// TwinCAT 3 PLC project Project_V25_Gr3
// ProgramVersion: 3.1.4026.13
// CompilerDefines: VISU_USEPROPERTYINFO
// libraries:
//   Tc2_Standard, * (Beckhoff Automation GmbH)
//   Tc2_System, * (Beckhoff Automation GmbH)
//   VisuDialogs, * (System)
// project tree:
//   / Engineer_HMI.TcVIS, GlobalTextList.TcGTLO, PlcTask.TcTTO, Visualization Manager.TcVMO (not stored)
//   Enums/ E_Status.TcDUT
//   Function Blocks/Currently not in use/ FB_EncoderScaling.TcPOU, FB_FeedForward.TcPOU (not stored), FB_Motion_Control.TcPOU, FB_SecondaryControlSinus.TcPOU, FB_SecondaryControlStartPos.TcPOU
//   Function Blocks/Deadband Comp/ FB_Deadband.TcPOU, FB_Deadband_Auto.TcPOU, FB_Deadband_Auto_sine.TcPOU
//   Function Blocks/Encoder_Payload/ FB_Encoder.TcPOU (not stored), FB_PayloadPosition.TcPOU
//   Function Blocks/FBs Auto Control/ FB_AutoSineMotion.TcPOU, FB_AutoStartPos.TcPOU, FB_Derivator.TcPOU, FB_SineActivation_SC.TcPOU
//   Function Blocks/FBs for Motion Control/Ekstra FBs/ FB_ControlReset_SC.TcPOU, FB_Feedforward_SC.TcPOU, FB_GainChooser.TcPOU (not stored), FB_Target_displacement.TcPOU
//   Function Blocks/FBs for Motion Control/ FB_Auto_Combination.TcPOU, FB_Auto_PC.TcPOU, FB_Auto_SC.TcPOU, FB_Enable_Motion.TcPOU, FB_EndStop.TcPOU, FB_Manual_PC.TcPOU, FB_Manual_SC.TcPOU, FB_MUX_selector.TcPOU, FB_Outputs.TcPOU
//   Function Blocks/ FB_Clock.TcPOU, FB_DisplacementControl.TcPOU, FB_DisplacementControl_SC.TcPOU, FB_DisplacementValveOutput.TcPOU, FB_Inputs.TcPOU, FB_Integrator.TcPOU, FB_Joystick.TcPOU, FB_StartPos.TcPOU, FB_StateMachine_Mode_Selection.TcPOU, FB_ValveOutput.TcPOU
//   Function Blocks/PIDgains/ FB_PIDgains.TcPOU
//   Function Blocks/Input_Scaling/ FB_JoystickInputScaling.TcPOU, FB_JoystickInputScaling_01.TcPOU (not stored), FB_PressureInputScaling.TcPOU (not stored), FB_Yoke_Input_Scaling.TcPOU (not stored)
//   Functions/ F_SineFunction_primary.TcPOU, F_SineFunction_secondary.TcPOU
//   GVLs/ G_IO.TcGVL, G_Motion_Control.TcGVL, G_Parameters.TcGVL, G_PID_Tuning.TcGVL, G_Sensors.TcGVL, G_Engineer_HMI.TcGVL
//   PIDs/ FB_PID_Controller.TcPOU, FB_PID_Controller_posref.TcPOU, FB_PID_controller_old.TcPOU, FB_PID_SC.TcPOU, FB_ResetIntegralController.TcPOU
//   POUs/ MAIN.TcPOU, P_MotionControl.TcPOU, P_Outputs.TcPOU
//   Structs/ ST_PressureInputScaling.TcDUT, ST_JoystickInputScaling.TcDUT, ST_Parameters.TcDUT, ST_ValveDeadBand.TcDUT, ST_ValveOutput.TcDUT, ST_YokeInputScaling.TcDUT
// real-time tasks:
//   TASK PlcTask: cycle T#10ms, priority 20, ADS port 350
// I/O:
//   DEVICE Device 1 (EtherCAT), AmsNetId 128.39.200.126.2.1
//     Term 1 (EK1200) [EK1200-5000 EtherCAT Power supply (2A E-Bus)]
//       Term 2 (EL1859) [EL1859 8Ch. Dig. Input 24V, 3ms, 8Ch. Dig. Output 24V, 0.5A]
//       Term 3 (EL3174) [EL3174 4Ch. Ana. Input +/-10V Diff., +/-20mA SingleEnded, 16 Bit]
//       Term 4 (EL4032) [EL4032 2Ch. Ana. Output +/-10V, 12bit]
//       Term 5 (EL3204) [EL3204 4Ch. Ana. Input PT100 (RTD)]
//       Term 6 (EK1110) [EK1110 EtherCAT extension]
//     Term 7 (EK1818) [EK1818 EtherCAT IO-Coupler  (1A E-Bus, 8 Ch. Dig. In, 3ms, 4 Ch. Dig. Out 24V, 0,5A)]
//       Term 8 (EL1008) [EL1008 8Ch. Dig. Input 24V, 3ms]
//       Term 9 (EL3174) [EL3174 4Ch. Ana. Input +/-10V Diff., +/-20mA SingleEnded, 16 Bit]
//       Term 10 (EL3068) [EL3068 8Ch. Ana. Input 0-10V]
//       Term 11 (EL4032) [EL4032 2Ch. Ana. Output +/-10V, 12bit]
//       Term 12 (EL4122) [EL4122 2Ch. Ana. Output  4-20mA, 16bit]
//       Term 14 (EL9011) [EL9011 End Terminal]
//     Box 13 (Fraba EtherCAT) [Absolute Rotary Encoder IXARC V01.05]
// variable links:
//   Project_V25_Gr3/Project_V25_Gr3 Instance <-> Device 1 (EtherCAT)/Box 13 (Fraba EtherCAT)
//     PlcTask Inputs/G_IO.nWinchEncoderValue <-> Encoder/Position Value
//   Project_V25_Gr3/Project_V25_Gr3 Instance <-> Device 1 (EtherCAT)/Term 7 (EK1818)
//     PlcTask Inputs/G_IO.bEmgOk <-> Channel 1/Input
//     PlcTask Outputs/G_IO.bEnablePCDV <-> Channel 10/Output
//     PlcTask Outputs/G_IO.bOpenBrakes <-> Channel 9/Output
//     PlcTask Outputs/G_IO.bWinchValveEnable <-> Channel 11/Output
//   Project_V25_Gr3/Project_V25_Gr3 Instance <-> Device 1 (EtherCAT)/Term 7 (EK1818)/Term 10 (EL3068)
//     PlcTask Inputs/G_IO.fJoyXraw <-> AI Standard Channel 6/Value
//     PlcTask Inputs/G_IO.fJoyYraw <-> AI Standard Channel 7/Value
//     PlcTask Inputs/G_IO.fJoyZraw <-> AI Standard Channel 8/Value
//     PlcTask Inputs/G_IO.fPressureReturn <-> AI Standard Channel 3/Value
//     PlcTask Inputs/G_IO.fPressureSupply <-> AI Standard Channel 2/Value
//     PlcTask Inputs/G_IO.fPressureWinchA <-> AI Standard Channel 1/Value
//     PlcTask Inputs/G_IO.fPressureWinchB <-> AI Standard Channel 4/Value
//   Project_V25_Gr3/Project_V25_Gr3 Instance <-> Device 1 (EtherCAT)/Term 7 (EK1818)/Term 11 (EL4032)
//     PlcTask Outputs/G_IO.fWinchPDCVOut <-> AO Outputs Channel 1/Analog output
//   Project_V25_Gr3/Project_V25_Gr3 Instance <-> Device 1 (EtherCAT)/Term 7 (EK1818)/Term 12 (EL4122)
//     PlcTask Outputs/G_IO.fWinchValveOut <-> Channel 1/Output
//   Project_V25_Gr3/Project_V25_Gr3 Instance <-> Device 1 (EtherCAT)/Term 7 (EK1818)/Term 8 (EL1008)
//     PlcTask Inputs/G_IO.bAutoSwitch <-> Channel 3/Input
//     PlcTask Inputs/G_IO.bDisplacementEnable <-> Channel 7/Input
//     PlcTask Inputs/G_IO.bManualSwitch <-> Channel 1/Input
//     PlcTask Inputs/G_IO.bOffSwitch <-> Channel 2/Input
//     PlcTask Inputs/G_IO.bStartButton <-> Channel 4/Input
//     PlcTask Inputs/G_IO.bStopButton <-> Channel 5/Input
//     PlcTask Inputs/G_IO.bWinchEnable <-> Channel 6/Input
//   Project_V25_Gr3/Project_V25_Gr3 Instance <-> Device 1 (EtherCAT)/Term 7 (EK1818)/Term 9 (EL3174)
//     PlcTask Inputs/G_IO.fPDCVMonitor <-> AI Standard Channel 1/Value
//     PlcTask Inputs/G_IO.fYoke <-> AI Standard Channel 4/Value
//     PlcTask Inputs/G_IO.nMoogMonitor <-> AI Standard Channel 2/Value

CONFIGURATION Project_V25_Gr3
    RESOURCE PLC ON TwinCAT3
        TASK PlcTask(INTERVAL := T#10ms, PRIORITY := 20);
        PROGRAM MAIN WITH PlcTask : MAIN;
    END_RESOURCE
END_CONFIGURATION

// ---- Enums/E_Status.TcDUT
{attribute 'qualified_only'}
{attribute 'strict'}
{attribute 'to_string'}
TYPE E_Status :
(
	Off,
	Fault,
	Ready,
	//Starting,
	Running,
	//Stopping,
	Checking
);
END_TYPE

// ---- Structs/ST_PressureInputScaling.TcDUT
TYPE ST_PressureInputScaling :
STRUCT
	fMaxInputValue 			: LREAL:= 32767.0;	// tunable max input value //   // denne verdien ble satt for å unngå å dele på 0, hvorfor må vi skrive det her men ikke i blueprint prosjekt
	fMinInputValue			: LREAL;	// tunable min input value  
	fMaxOutputValue  		: LREAL;	// max sensor output value
	fMinOutputValue  		: LREAL;	// min sensor output value	
END_STRUCT
END_TYPE

// ---- Structs/ST_JoystickInputScaling.TcDUT
TYPE ST_JoystickInputScaling :
STRUCT
	fMaxInputValue			: LREAL;	// tunable max input value
	fMinInputValue 			: LREAL;	// tunable min input value
	fNeutralInputValue  	: LREAL;	// tunable neutral input value
	fNeutralDeadband		: LREAL;	// tunable dead_band value
	fMaxOutputValue  		: LREAL;	// normalized max output value
	fMinOutputValue  		: LREAL;	// normalized min output value
	fNeutralOutputValue  	: LREAL;	// normalized neutral output value
END_STRUCT
END_TYPE

// ---- Structs/ST_Parameters.TcDUT
 TYPE ST_Parameters : // Blir gjort globale i GVL
STRUCT
	fCyclicTime 					: LREAL := 0.01; // [s]
	fMaxWinchVelocityLimit 			: LREAL := 0.25; // [m/s] Blueprint: 0.025
	fMaxWinchVelocityLimit_SC		: LREAL := 0.25;
	bWinchDeadBandCompOn 			: BOOL := FALSE;
	bDisplacementDeadBandCompOn 	: BOOL := FALSE;
	stWinchValveDeadBand 			: ST_ValveDeadBand := (fPosMax := 32767.0, fPosMin := 16383.0, fNegMin := 16383.0, fNegMax := 0.0);
	stDisplacementValveDeadBand 	: ST_ValveDeadBand := (fPosMax := 10000.0, fPosMin := 450.0, fNegMin := 450.0, fNegMax := 10000.0);
	stPressureSensorScaling400bar 	: ST_PressureInputScaling := (fMaxInputValue := 32767.0, fMinInputValue := 0.0, fMaxOutputValue := 400.0, fMinOutputValue := 0.0);
	stPressureSensorScaling40bar 	: ST_PressureInputScaling := (fMaxInputValue := 32767.0, fMinInputValue := 0.0, fMaxOutputValue := 40.0, fMinOutputValue := 0.0);
	stJoystickInputScalingX 		: ST_JoystickInputScaling := (fMaxInputValue := 14790.0, fMinInputValue := 1797.0, fNeutralInputValue := 8400, fNeutralDeadband := 50.0, fMaxOutputValue := 1.0, fMinOutputValue := 0.0, fNeutralOutputValue := 0.5);
	stJoystickInputScalingY 		: ST_JoystickInputScaling := (fMaxInputValue := 14770.0, fMinInputValue := 1829.0, fNeutralInputValue := 8340, fNeutralDeadband := 50.0, fMaxOutputValue := 1.0, fMinOutputValue := -1.0, fNeutralOutputValue := 0.0);
	stJoystickInputScalingZ 		: ST_JoystickInputScaling := (fMaxInputValue := 14830.0, fMinInputValue := 1804.0, fNeutralInputValue := 8380, fNeutralDeadband := 50.0, fMaxOutputValue := 1.0, fMinOutputValue := -1.0, fNeutralOutputValue := 0.0);
	fWinchEncoderOffset 			: LREAL := 12814.994735637447; // Encoder value at zero (Cylinder out / second layaer)
	stYokeInputScaling 				: ST_YokeInputScaling := (fMaxInputValue := 25000.0, fMinInputValue := 6150.0, fNeutralInputValue := 15470, fNeutralDeadband := 0.0, fMaxOutputValue := 1.0, fMinOutputValue := -1.0, fNeutralOutputValue := 0.0);
	fWinchDrumRadius 				: LREAL := 0.075;
	fWinchEndStopPos 				: LREAL := 3.0;
	fWinchEndStopPos_soft			: LREAL := 2.55;
	fWinchEndStopNeg 				: LREAL := 0.05;
	fWinchEndStopNeg_soft			: LREAL := 0.25;
	fPayloadMass 					: LREAL := 78.0;
	
	
END_STRUCT
END_TYPE

// ---- Structs/ST_ValveDeadBand.TcDUT
TYPE ST_ValveDeadBand :
STRUCT
	fPosMax	: LREAL; // Positive min value [19660..29490]
	fPosMin	: LREAL; // Positive max value [19660..29490]
	fNegMin : LREAL; // Negative max value [9830..19660]
	fNegMax	: LREAL; // Negative min value [9830..19660]
END_STRUCT
END_TYPE

// ---- Structs/ST_ValveOutput.TcDUT
TYPE ST_ValveOutput :
STRUCT
	bEnable					AT %Q* : BOOL := 0;
	nValveOutput 			AT %Q* : INT := 19660;
END_STRUCT
END_TYPE

// ---- Structs/ST_YokeInputScaling.TcDUT
TYPE ST_YokeInputScaling :
STRUCT
	fMaxInputValue			: LREAL;	// tunable max input value
	fMinInputValue 			: LREAL;	// tunable min input value
	fNeutralInputValue  	: LREAL;	// tunable neutral input value
	fNeutralDeadband		: LREAL;	// tunable dead_band value
	fMaxOutputValue  		: LREAL;	// normalized max output value
	fMinOutputValue  		: LREAL;	// normalized min output value
	fNeutralOutputValue  	: LREAL;	// normalized neutral output value
END_STRUCT
END_TYPE

// ---- GVLs/G_IO.TcGVL
{attribute 'qualified_only'}
VAR_GLOBAL
	// Digitale inputs
	bEmgOk 			     AT %I* : BOOL; 
	bStartButton 	     AT %I* : BOOL;
	bStopButton 	     AT %I* : BOOL; 
	bOffSwitch		     AT %I* : BOOL;  
	bManualSwitch	     AT %I* : BOOL; 
	bAutoSwitch		 	 AT %I* : BOOL; 
	bWinchEnable 		 AT %I* : BOOL; 
	bDisplacementEnable  AT %I* : BOOL;
	
	// Analoge Intputs
	fJoyXraw 			 AT %I* : INT; 
	fJoyYraw			 AT %I* : INT; 
	fJoyZraw 			 AT %I* : INT; 
	fPDCVMonitor		 AT %I* : INT; 
	nMoogMonitor		 AT %I* : INT; 
	fYoke				 AT %I* : INT; 
	fPressureWinchA 	 AT %I* : INT; 
	fPressureWinchB 	 AT %I* : INT; 
	fPressureSupply 	 AT %I* : INT; 
	fPressureReturn 	 AT %I* : INT; 
	nWinchEncoderValue	 AT %I* : UDINT; 
	
	// Digitale Outputs
	bOpenBrakes 		 AT %Q* : BOOL; 
	bEnablePCDV 		 AT %Q* : BOOL; 
	bWinchValveEnable 	 AT %Q* : BOOL; 
	
	// Analoge Outputs
	fWinchPDCVOut 		 AT %Q* : INT := 10000; 
	fWinchValveOut 		 AT %Q* : INT := 16383; 
	
	// New Test
	bTestNew AT %I* : BOOL;
	nTestNew AT %I* : INT;
	OutTestNew AT %Q* : BOOL;
	
END_VAR

// ---- GVLs/G_Motion_Control.TcGVL
{attribute 'qualified_only'}
VAR_GLOBAL
	//////////Primary Control/////////
//AutoStartPos
fWinchValveNormalizedInput 					: LREAL;	
bOpenBreak									: BOOL;

//AutoSineMotion
fWinchValveNormalizedInput_sine 			: LREAL;
fSineReferenceSignal						: LREAL;

// Position Errors
fPosition_error_SineMotion 					: LREAL; 
fPosition_error_StartPos					: LREAL;

//Displacement Sine
fDisplacementControlSignal_sine				: LREAL;

//Manual joystick posref
fWinchPosRefManual							: LREAL; //to make it a global variable for plotting 
fWinchValveInput_joystick_posref			: LREAL;



//////// Secondary control////////
fWinchPosRefManual_secondary				: LREAL;
fSCVInput_joystick_posref_secondary			: LREAL;

//Auto Sine Motion SC
fSineRefSignal_SC							: LREAL;
fVelRef_Sine_SC								: LREAL;

//Outer and inner loop sequence SC
fOutPutSignal_OL							: LREAL; //Skrive manual bak disse og oppdatere OPC UA
fDeadbandComp_out							: LREAL;

//Ikke lagt til i OPC UA
fOutPutSignal_OL_Auto						: LREAL;
fDeadbandComp_out_Auto						: LREAL;

//Ikke i bruk
fPosition_error_StartDisplacement 			: LREAL; 
fDisplacementControlSignal_Secondary		: LREAL;
bOpenBreak_Secondary						: BOOL;
END_VAR

// ---- GVLs/G_Parameters.TcGVL
{attribute 'qualified_only'}
VAR_GLOBAL
stParam		:	ST_Parameters;
END_VAR

// ---- GVLs/G_PID_Tuning.TcGVL
{attribute 'qualified_only'}
VAR_GLOBAL
	/////////Primary control/////////
	
	//MOOG valve
	fProportinalGain_output_MOOG 		: LREAL;
	fIntegralGain_output_MOOG			: LREAL;
	fDerivateGain_output_MOOG 			: LREAL;
	PID_output_MOOG						: LREAL;
	
	//Manual Control joystick pos ref
	fProportinalGain_output_joypos 		: LREAL;
	fIntegralGain_output_joypos			: LREAL;
	fDerivateGain_output_joypos 		: LREAL;
	ferror_joypos 						: LREAL;
	
	/////////Secondary control//////
	
	//Displacement control
	fYoke_error 						: LREAL;
	fPout_IL					 		: LREAL;
	fIout_IL					 		: LREAL;
	fDout_IL					 		: LREAL;
	PID_output_IL						: LREAL;
	Int_error_threshold					: LREAL := 0.0001;
	
	//Manual Control joystick posref secondary
	fPout_OL							: LREAL;
	fIout_OL							: LREAL;
	fDout_OL							: LREAL;
	fPout_OL_Auto							: LREAL;
	fIout_OL_Auto							: LREAL;
	fDout_OL_Auto							: LREAL;
	fPout_OL_Auto_sine							: LREAL;
	fIout_OL_Auto_sine							: LREAL;
	fDout_OL_Auto_sine							: LREAL;
	
	ferror_OL							: LREAL; //Skrive manual bak denne
	ferror_OL_Auto_startpos				: LREAL;
	ferror_OL_Auto_sine					: LREAL;
	
	
	////Combination////
	fPout_OL_combi							: LREAL;
	fIout_OL_combi							: LREAL;
	fDout_OL_combi							: LREAL;
	ferror_OL_combi							: LREAL;
	
END_VAR

// ---- GVLs/G_Sensors.TcGVL
{attribute 'qualified_only'}
VAR_GLOBAL
	fJoystickNormalizedY 					: LREAL; 
	fJoystickNormalizedX 					: LREAL; 
	fJoystickNormalizedZ 					: LREAL; 
	fYokeNormalizedFeedback 				: LREAL; 
	fPressureWinchA 	 					: LREAL; 
	fPressureWinchB 	 					: LREAL; 
	fPressureSupply 	 					: LREAL; 
	fPressureReturn 	 					: LREAL; 
	fWinchEncoderPosition 					: LREAL;
	fWinchEncoderPositionNormalized 		: LREAL;
	fPayLoadPosition 						: LREAL;
	fDeltaPMotor 							: LREAL;
	
	//Egentlig en Output/ NEIUNEI
	fWinchValveOutNormalized				: LREAL;
END_VAR

// ---- GVLs/G_Engineer_HMI.TcGVL
{attribute 'qualified_only'}
VAR_GLOBAL
	
//////////PID GAINS//////////

////Primary Control//////
// PID Manual control joystick pos ref Primary
	
	bPID_enable_JoyPosref_PC		: BOOL := TRUE;
	bPgain_enable_joy_posref		: BOOL := TRUE;
	bIgain_enable_joy_posref		: BOOL;
	bPgain_joy_posref_write			: BOOL;
	bIgain_joy_posref_write			: BOOL;
	bDgain_joy_posref_write			: BOOL;
	
	fPGain_JoyPosref_PC 			: LREAL;
	fIGain_JoyPosref_PC				: LREAL;
	fDGain_JoyPosref_PC				: LREAL;

// PID MOOG Valve (Auto PC)
	fPgain_MOOG						: LREAL;
	bPenable_MOOG					: BOOL := TRUE; //Ønsker P ledd på fra start
	bPgain_MOOG_write				: BOOL;
	
	fIgain_MOOG 					: LREAL; 
	bIenable_MOOG 					: BOOL;
	bIgain_MOOG_write				: BOOL; 

////// Secondary Control ////////

// PID Outer loop 
bPID_enable_OL					: BOOL := TRUE;

fPGain_OL_Pos					: LREAL;
fPGain_OL_Neg					: LREAL;
bPenable_OL						: BOOL := TRUE;
bPGain_OL_write_pos				: BOOL;
bPGain_OL_write_neg				: BOOL;

fIGain_OL_Pos					: LREAL;
fIGain_OL_Neg					: LREAL;
bIenable_OL						: BOOL;
bIGain_OL_write_pos				: BOOL;
bIGain_OL_write_neg				: BOOL;

// PID Inner loop
bPID_enable_IL					: BOOL := TRUE;

fPGain_IL_Pos					: LREAL;
fPGain_IL_Neg					: LREAL;
bPenable_IL						: BOOL := TRUE;
bPGain_IL_write_pos				: BOOL;
bPGain_IL_write_neg				: BOOL;

fIGain_IL_Pos					: LREAL;
fIGain_IL_Neg					: LREAL;
bIenable_IL						: BOOL;
bIGain_IL_write_pos				: BOOL;
bIGain_IL_write_neg				: BOOL;

fDGain_IL_Pos					: LREAL;
fDGain_IL_Neg					: LREAL;
bDenable_IL						: BOOL;
bDGain_IL_write_pos					: BOOL;
bDGain_IL_write_neg					: BOOL;



////////// PID GAINS End ///////////////////


	//Control chooser
	bPrimary_Control				: BOOL;	
	bPrimary_Control_active			: BOOL := FALSE;
	bSecondary_Control				: BOOL;
	bSecondary_Control_active		: BOOL := FALSE;

	//Endstop
	bEndStopUpActive 				: BOOL;
	bEndStopDownActive 				: BOOL;
	bEndStopOverride 				: BOOL; 
	
	/////Primary Control//////
	bManualControl_enable			: BOOL;
	
	
	
	// Auto Start Pos
	bAutoStartPosEnable				: BOOL;
	fAutoStartPos_target			: LREAL := 1.4;
	
	// Auto Sine Motion
	bAutoSineMotionEnable			 : BOOL; 
	
	// Displacement Sine Wave control: 
	bSineDisplacement				 : BOOL; 
	
	//Sine wave parameters
	fAmp 							: LREAL := 0.2;
	fFreq 							: LREAL := 0.1;
	fSinemidpoint					: LREAL := 1.4;
	ft_ENV							: LREAL := 10.0;
	
	
	
	
///// Primary Control End///////	
	
	
////// Secondary Control///////
	
//Displacementcontrol 
	bDisplacement_target_active		: BOOL;
	fDisplacement_target			: LREAL := 1.0;
	bJoystick_slider_active			: BOOL;
	bSecondaryStartPosEnable 		: BOOL;
	fSecondaryStartPos_target		: LREAL := 1.4;
	bSecondarySineMotionEnable		: BOOL;


	
	//Integral reset (antiwindup)
	fMaxerror_dis					: LREAL;
	
	
//PID Gains for Manual control joystick posref
	
	bManual_Secondary_joyposref_enable	: BOOL := TRUE;
	
// Deadband compensation (gjort om til var persistants som ligger i FB_PIDgains)
fUpperdeadband						: LREAL;
fNeutraldeadband					: LREAL;
fLowerdeadband						: LREAL;
bUpperWrite							: BOOL;
bNeutralWrite						: BOOL;
bLowerWrite							: BOOL;
	
////////Primary and Secondary combination//////
bCombinationActive					: BOOL;
bAutoSineCombi						: BOOL;

	
//StepInput displacement ikke lagt inn etter å ha ryddet, kan legges inn i 
//Manual SC om det trengs (la tidligere i P_outputs
bStepInput								: BOOL;
bStartStepInput							: BOOL;
fStepInput								: LREAL;
fDuration								: LREAL;

	
END_VAR

// ---- POUs/MAIN.TcPOU
PROGRAM MAIN
VAR
	bFunction_Blocks_enable				: BOOL := TRUE;
	fb_StateMachine_Mode_Selection	 	: FB_StateMachine_Mode_Selection;
	fb_Joystick_input_Scaling			: FB_JoystickInputScaling;
	fb_Joystick							: FB_Joystick;
	fb_ValveOutput						: FB_ValveOutput;
	fb_Encoder							: FB_Encoder; 
	fb_PressureInputScaling 			: FB_PressureInputScaling;
	fb_PayloadPosition					: FB_PayloadPosition;
	fb_Inputs							: FB_Inputs;
	eStatus								: E_Status;
	
	fbPIDgains							: FB_PIDgains;
END_VAR

P_MotionControl();

IF bFunction_Blocks_enable THEN
	fb_StateMachine_Mode_Selection();
	fb_Joystick_input_Scaling();
	fb_Joystick();
	fb_ValveOutput();
	fb_Encoder();
	fb_PressureInputScaling();
	fb_PayloadPosition();
	fb_Inputs();
	
	fbPIDgains();
END_IF

//Update eStatus
fb_StateMachine_Mode_Selection(
	eStatus => eStatus
	);
//	eStatus := E_Status.Running;
	
	

////////Select Primary eller Secondary control//////////////
IF G_Engineer_HMI.bPrimary_Control THEN
	G_Engineer_HMI.bPrimary_Control_active := TRUE;
	G_Engineer_HMI.bSecondary_Control_active := FALSE;
ELSIF G_Engineer_HMI.bSecondary_Control THEN
	G_Engineer_HMI.bPrimary_Control_active := FALSE;
	G_Engineer_HMI.bSecondary_Control_active := TRUE;
END_IF

END_PROGRAM

// ---- Function Blocks/FB_StateMachine_Mode_Selection.TcPOU
FUNCTION_BLOCK FB_StateMachine_Mode_Selection
VAR_INPUT
END_VAR
VAR_OUTPUT
eStatus : E_Status := E_Status.Checking; //Er dette til for å definere utgangen, kunne vi brukt structen (Enumen) direkte i koden?
END_VAR
VAR
	
	bStatusOk : BOOL; // Control variable 
	bFault : BOOL := FALSE;
	//bRunning : BOOL := TRUE; ikke nødvendig
END_VAR

	// State Machine for mode selection - Off, Fault, Ready, Running and Checking 
	
	// Variable bStatusOk, used troughout the function: 
IF G_IO.bEmgOk AND NOT(G_IO.bStopButton) AND NOT(G_IO.bOffSwitch) AND NOT(bFault) THEN 
	bStatusOk := TRUE;
ELSE 
	bStatusOk := FALSE;
END_IF

CASE eStatus OF
	E_Status.Checking: // Checking state (initially here)
	  IF bFault THEN
         eStatus := E_Status.Fault; 
	  END_IF
	  
	  IF bStatusOk THEN 
		  eStatus := E_Status.Ready;
	  END_IF
	  
	  IF NOT bStatusOk THEN
		 eStatus := E_Status.Off;
	  END_IF
	  
	 E_Status.Off:
	   IF bStatusOk THEN
			eStatus := E_Status.Checking;
	END_IF
		
	IF bFault THEN
			eStatus := E_Status.Fault;
	END_IF
		
	  E_Status.Fault:
		  IF NOT bFault THEN
			  eStatus := E_Status.Checking;
		  END_IF
		  
	E_Status.Ready:
	  IF G_IO.bStartButton AND bStatusOk THEN 
		  eStatus := E_Status.Running;
	  END_IF
	  
	  IF NOT(bStatusOk) OR bFault THEN
		  eStatus := E_Status.Checking;
	  END_IF
	  
	E_Status.Running: 
	
	 IF NOT(bStatusOk) OR bFault THEN 
		 eStatus := E_Status.Checking;
	 END_IF
	 
	 ELSE 
		 eStatus := E_Status.Checking;
  END_CASE

END_FUNCTION_BLOCK

// ---- Function Blocks/Input_Scaling/FB_JoystickInputScaling.TcPOU
FUNCTION_BLOCK FB_JoystickInputScaling
VAR_INPUT
	bEnable 				: BOOL;
	nRawInput 				: INT;
	stJoystickInputScaling  : ST_JoystickInputScaling;
END_VAR
VAR_OUTPUT
	fNormalizedOutput 		: LREAL;
END_VAR
VAR
	fRawInput 				: LREAL;
	fTempInput 				: LREAL;
	fTempOutput 			: LREAL;
END_VAR

fRawInput := INT_TO_LREAL(nRawInput);

fTempInput := fRawInput - stJoystickInputScaling.fNeutralInputValue;

IF fTempInput > stJoystickInputScaling.fNeutralDeadband THEN
	fTempOutput := fTempInput/(stJoystickInputScaling.fMaxInputValue - stJoystickInputScaling.fNeutralInputValue);
ELSIF fTempInput < -stJoystickInputScaling.fNeutralDeadband THEN	
	fTempOutput := fTempInput/(stJoystickInputScaling.fNeutralInputValue - stJoystickInputScaling.fMinInputValue);
ELSE
	fTempOutput := 0.0;
END_IF

IF NOT(bEnable) THEN
	fNormalizedOutput := 0.0;
ELSE
	fNormalizedOutput := LIMIT(stJoystickInputScaling.fMinOutputValue, fTempOutput, stJoystickInputScaling.fMaxOutputValue);
END_IF

END_FUNCTION_BLOCK

// ---- Function Blocks/FB_Joystick.TcPOU
FUNCTION_BLOCK FB_Joystick
VAR_INPUT
	bEnable 			: BOOL;
	fNormalizedInput 	: LREAL;
	stParam 			: ST_Parameters;
END_VAR
VAR_OUTPUT
	fOuput : LREAL;
END_VAR
VAR
END_VAR

IF bEnable THEN
	
	fOuput := fNormalizedInput*G_Parameters.stParam.fMaxWinchVelocityLimit_SC;
ELSE
	fOuput := 0.0;
END_IF

END_FUNCTION_BLOCK

// ---- Function Blocks/FB_ValveOutput.TcPOU
FUNCTION_BLOCK FB_ValveOutput
VAR_INPUT
	bEnable : BOOL; 
	bDeadBandCompOn : BOOL;
	stValveDeadBand : ST_ValveDeadBand; 
	fNormalizedInput : LREAL; 
END_VAR
VAR_OUTPUT
	bEnableValveOutput : BOOL; 
	nOutput : INT; 
END_VAR
VAR
	nOffset 	: INT := 16383; // KVIFOR
	nMaxValue	: INT := 20000;
	nMinValue 	: INT :=  12766;
	nTempOutput : INT := 16383;
END_VAR

//To måter er satt opp, kan endres i Engineer_HMI. En er satte parametere, den andre er parametere fra struct
IF bDeadBandCompOn THEN
	IF fNormalizedInput > 0.0 THEN
		nTempOutput := LREAL_TO_INT(ABS(fNormalizedInput*(stValveDeadBand.fPosMax - stValveDeadBand.fPosMin) + stValveDeadBand.fPosMin));
	ELSIF fNormalizedInput < 0.0 THEN 
		nTempOutput := LREAL_TO_INT(ABS(fNormalizedInput*(stValveDeadBand.fNegMax - stValveDeadBand.fNegMin) - stValveDeadBand.fNegMin));	
	ELSE 
		nTempOutput := nOffset;	//Offset ses som 0 (nøytral), fordi signalet går fra 0 til 32767.												
	END_IF

ELSE 
	IF fNormalizedInput > 0.0  THEN
		//Gjør om inputen mellom 0 og 1 til en output mellom 16383 (nøytral) og 32767(max)
		nTempOutput := LREAL_TO_INT(ABS(fNormalizedInput*(32767.0 - 16383.0) + 16383.0)); //ABS må til fordi output er en positiv verdi mellom 0 og 32767
	ELSIF fNormalizedInput < 0.0  THEN
		//Gjør om inputen mellom 0 og -1 til en output mellom 0 (min) og 16383 (nøytral)
		nTempOutput := LREAL_TO_INT(ABS(fNormalizedInput*(0 - 16383.0) - 16383.0));
	ELSE
		nTempOutput := nOffset; //Her settes også verdien til nøytral om det ikke er noen input
	END_IF	
	
END_IF

//Om den er enabled blir verdien sendt ut
IF bEnable THEN
	
	nOutput := LIMIT(nMinValue, nTempOutput, nMaxValue);
	bEnableValveOutput := TRUE;
//Eller så sender den ut nøytral verdi
ELSE 
	nOutput := nOffset;
	bEnableValveOutput := FALSE;
END_IF

END_FUNCTION_BLOCK

// ---- Function Blocks/Encoder_Payload/FB_PayloadPosition.TcPOU
FUNCTION_BLOCK FB_PayloadPosition
VAR_INPUT
END_VAR
VAR_OUTPUT
END_VAR
VAR
END_VAR

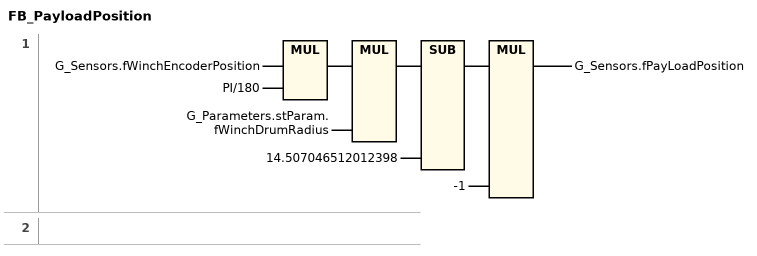
// NETWORK 1
G_Sensors.fPayLoadPosition := ((G_Sensors.fWinchEncoderPosition * (PI/180)) * G_Parameters.stParam.fWinchDrumRadius - 14.507046512012398) * -1;

// NETWORK 2

END_FUNCTION_BLOCK

// ---- Function Blocks/FB_Inputs.TcPOU
FUNCTION_BLOCK FB_Inputs 
VAR_INPUT
	fbJoystickWinch : FB_JoystickInputScaling; 
	fbJoystickRot : FB_JoystickInputScaling; 
	fbYokeInputScaling : FB_Yoke_Input_Scaling;
	fbWinchPosition : FB_Encoder;
	fbPressureSupply : FB_PressureInputScaling; 
	fbPressureReturn : FB_PressureInputScaling;
	fbPressureWinch_A_Input : FB_PressureInputScaling;
	fbPressureWInch_B_Input : FB_PressureInputScaling; 
END_VAR
VAR_OUTPUT
END_VAR
VAR
END_VAR

fbJoystickWinch(
	bEnable := G_IO.bAutoSwitch OR G_IO.bManualSwitch,
	nRawInput := G_IO.fJoyYraw, 
	stJoystickInputScaling := G_Parameters.stParam.stJoystickInputScalingY, 
	fNormalizedOutput => G_Sensors.fJoystickNormalizedY
);

fbJoystickRot(
	bEnable := G_IO.bManualSwitch, 
	nRawInput := G_IO.fJoyZraw,
	stJoystickInputScaling := G_Parameters.stParam.stJoystickInputScalingZ,
    fNormalizedOutput => G_Sensors.fJoystickNormalizedZ
);

fbYokeInputScaling(
	bEnable := TRUE, //Vil lese Yokeverdi hele tiden så den settes til TRUE (var G_IO.bManualSwitch før)
	nRawInput := G_IO.fYoke, 
	stYokeInputScaling := G_Parameters.stParam.stYokeInputScaling,
	fNormalizedOutput => G_Sensors.fYokeNormalizedFeedback
);

fbWinchPosition(
nRawInput := G_IO.nWinchEncoderValue,
fEncoderOffset := G_Parameters.stParam.fWinchEncoderOffset,
fPosition => G_Sensors.fWinchEncoderPosition
);

fbPressureSupply(
	nRawInput := G_IO.fPressureSupply,
	stPressureInputScaling := G_Parameters.stParam.stPressureSensorScaling400bar,
	fOutput => G_Sensors.fPressureSupply
);

fbPressureReturn(
	nRawInput := G_IO.fPressureReturn,
	stPressureInputScaling := G_Parameters.stParam.stPressureSensorScaling40bar,
	fOutput => G_Sensors.fPressureReturn
	);
	
fbPressureWinch_A_Input(
	nRawInput := G_IO.fPressureWinchA, 
	stPressureInputScaling := G_Parameters.stParam.stPressureSensorScaling400bar, 
	fOutput => G_Sensors.fPressureWinchA
	);
	
fbPressureWinch_B_Input(
nRawInput := G_IO.fPressureWinchB,
stPressureInputScaling := G_Parameters.stParam.stPressureSensorScaling400bar, 
fOutput => G_Sensors.fPressureWinchB
);

// Trykkfall over motor: 

G_Sensors.fDeltaPMotor := (G_Sensors.fPressureWinchA - G_Sensors.fPressureWinchB);

END_FUNCTION_BLOCK

// ---- Function Blocks/PIDgains/FB_PIDgains.TcPOU
FUNCTION_BLOCK FB_PIDgains
VAR_INPUT
END_VAR
VAR_OUTPUT
END_VAR

VAR PERSISTENT
	
	/////Primary Control/////
	
	//Joystick Posref
	fPGain_JoyPosref_PC 				: LREAL;
	fIGain_JoyPosref_PC					: LREAL;
	fDGain_JoyPosref_PC					: LREAL;
	
	
	//Auto PC
	fPGain_MOOG							: LREAL;
	fIGain_MOOG							: LREAL;
	
	/////Secondary Control////
	
	//Outer loop
	fPGain_OL_Pos					: LREAL;
	fIGain_OL_Pos					: LREAL;
	fPGain_OL_Neg					: LREAL;
	fIGain_OL_Neg					: LREAL;
	
	//Inner loop
	fPGain_IL_Pos					: LREAL;
	fIGain_IL_Pos					: LREAL;
	fPGain_IL_Neg					: LREAL;
	fIGain_IL_Neg					: LREAL;
	fDGain_IL_Pos					: LREAL;
	fDGain_IL_Neg					: LREAL;
	
	/////Deadband Compensation/////
	fUpper							: LREAL;
	fNeutral						: LREAL;
	fLower							: LREAL;
	
END_VAR

VAR
END_VAR

	
	/////Primary Control/////
	
	//Joystick Posref
IF NOT(G_Engineer_HMI.bPgain_joy_posref_write) THEN
	G_Engineer_HMI.fPGain_JoyPosref_PC := fPGain_JoyPosref_PC; //Update to the persistent variable
ELSE
	fPGain_JoyPosref_PC := G_Engineer_HMI.fPGain_JoyPosref_PC; //Connect the gain to the global HMI
END_IF
	
	
IF NOT(G_Engineer_HMI.bIgain_joy_posref_write) THEN
	G_Engineer_HMI.fIGain_JoyPosref_PC := fIGain_JoyPosref_PC; //Update to the persistent variable
ELSE
	fIGain_JoyPosref_PC := G_Engineer_HMI.fIGain_JoyPosref_PC; //Connect the gain to the global HMI
END_IF
	
	
IF NOT(G_Engineer_HMI.bDgain_joy_posref_write) THEN
	G_Engineer_HMI.fDGain_JoyPosref_PC := fDGain_JoyPosref_PC; //Update to the persistent variable
ELSE
	fDGain_JoyPosref_PC := G_Engineer_HMI.fDGain_JoyPosref_PC; //Connect the gain to the global HMI
END_IF
	
	//Auto PC
IF NOT(G_Engineer_HMI.bPgain_MOOG_write) THEN
	G_Engineer_HMI.fPgain_MOOG := fPGain_MOOG; 
ELSE
	fPGain_MOOG := G_Engineer_HMI.fPgain_MOOG;
END_IF


IF NOT(G_Engineer_HMI.bIgain_MOOG_write) THEN
	G_Engineer_HMI.fIgain_MOOG := fIGain_MOOG;
ELSE
	fIGain_MOOG := G_Engineer_HMI.fIgain_MOOG;
END_IF	


//////// Secondary Control /////////

//Outer loop
//Positive
IF NOT(G_Engineer_HMI.bPGain_OL_write_pos) THEN
	G_Engineer_HMI.fPGain_OL_Pos := fPGain_OL_Pos; 
ELSE
	fPGain_OL_Pos := G_Engineer_HMI.fPGain_OL_Pos;
END_IF


IF NOT(G_Engineer_HMI.bIGain_OL_write_pos) THEN
	G_Engineer_HMI.fIGain_OL_Pos := fIGain_OL_Pos;
ELSE
	fIGain_OL_Pos := G_Engineer_HMI.fIGain_OL_Pos;
END_IF	

//Negative
IF NOT(G_Engineer_HMI.bPGain_OL_write_neg) THEN
	G_Engineer_HMI.fPGain_OL_Neg := fPGain_OL_Neg; 
ELSE
	fPGain_OL_Neg := G_Engineer_HMI.fPGain_OL_Neg;
END_IF


IF NOT(G_Engineer_HMI.bIGain_OL_write_neg) THEN
	G_Engineer_HMI.fIGain_OL_Neg := fIGain_OL_Neg;
ELSE
	fIGain_OL_Neg := G_Engineer_HMI.fIGain_OL_Neg;
END_IF	


//Inner loop
//Positive
IF NOT(G_Engineer_HMI.bPGain_IL_write_pos) THEN
	G_Engineer_HMI.fPGain_IL_Pos := fPGain_IL_Pos; 
ELSE
	fPGain_IL_Pos := G_Engineer_HMI.fPGain_IL_Pos;
END_IF


IF NOT(G_Engineer_HMI.bIGain_IL_write_pos) THEN
	G_Engineer_HMI.fIGain_IL_Pos := fIGain_IL_Pos;
ELSE
	fIGain_IL_Pos := G_Engineer_HMI.fIGain_IL_Pos;
END_IF	

IF NOT(G_Engineer_HMI.bDGain_IL_write_pos) THEN
	G_Engineer_HMI.fDGain_IL_Pos := fDGain_IL_Pos;
ELSE
	fDGain_IL_Pos := G_Engineer_HMI.fDGain_IL_Pos;
END_IF	

//Negative
IF NOT(G_Engineer_HMI.bPGain_IL_write_neg) THEN
	G_Engineer_HMI.fPGain_IL_Neg := fPGain_IL_Neg; 
ELSE
	fPGain_IL_Neg := G_Engineer_HMI.fPGain_IL_Neg;
END_IF


IF NOT(G_Engineer_HMI.bIGain_IL_write_neg) THEN
	G_Engineer_HMI.fIGain_IL_Neg := fIGain_IL_Neg;
ELSE
	fIGain_IL_Neg := G_Engineer_HMI.fIGain_IL_Neg;
END_IF	

IF NOT(G_Engineer_HMI.bDGain_IL_write_neg) THEN
	G_Engineer_HMI.fDGain_IL_Neg := fDGain_IL_Neg;
ELSE
	fDGain_IL_Neg := G_Engineer_HMI.fDGain_IL_Neg;
END_IF	

/////////Deadband Compensation////////////
IF NOT(G_Engineer_HMI.bUpperWrite) THEN
	G_Engineer_HMI.fUpperdeadband := fUpper;
ELSE
	fUpper := G_Engineer_HMI.fUpperdeadband;
END_IF

IF NOT(G_Engineer_HMI.bNeutralWrite) THEN
	G_Engineer_HMI.fNeutraldeadband := fNeutral;
ELSE
	fNeutral := G_Engineer_HMI.fNeutraldeadband;
END_IF

IF NOT(G_Engineer_HMI.bLowerWrite) THEN
	G_Engineer_HMI.fLowerdeadband:= fLower;
ELSE
	fLower := G_Engineer_HMI.fLowerdeadband;
END_IF

END_FUNCTION_BLOCK

// ---- POUs/P_MotionControl.TcPOU
PROGRAM P_MotionControl
VAR
	

//////Dette brukes i det nye////////////

//Enable Motion
	bAutoEnable_PC 							: BOOL;
	bManualEnable_PC 						: BOOL; 
	bAutoEnable_SC 							: BOOL; 
	bManualEnable_SC					    : BOOL;
	bCombinationEnable						: BOOL;

/////////// Function blocks////////// 
	
	//Enable Motion
	fbEnableMotion							: FB_Enable_Motion;
	
	//Primary Control
	fbManual_PC								: FB_Manual_PC;
	fbAuto_PC								: FB_Auto_PC;
	
	//Secondary Control
	fbManual_SC								: FB_Manual_SC;
	fbAuto_SC								: FB_Auto_SC;

	//Combination
	fbCombination							: FB_Auto_Combination;

	//Endstop
	fbEndstop								: FB_EndStop;

	//MUX
	fbMUX_selector							: FB_MUX_selector;

/////OutPut Variables////
	fPCV_MPC							: LREAL;
	fSCV_MPC							: LREAL;
	
	fPCV_APC							: LREAL;
	fSCV_APC							: LREAL;
	
	fPCV_MSC							: LREAL;
	fSCV_MSC							: LREAL;
	
	fPCV_ASC							: LREAL;
	fSCV_ASC							: LREAL;
	
	fPCV_combi							: LREAL;
	fSCV_combi							: LREAL;
	
	//After MUX
	fPCV							: LREAL;
	fSCV							: LREAL;
	fPCV_norm_input					: LREAL;
	fSCV_norm_input					: LREAL;
	
	
//ValveOutputs
fbOutputs							: FB_Outputs;
fPCV_raw							: INT;
fSCV_raw							: INT;
	
END_VAR

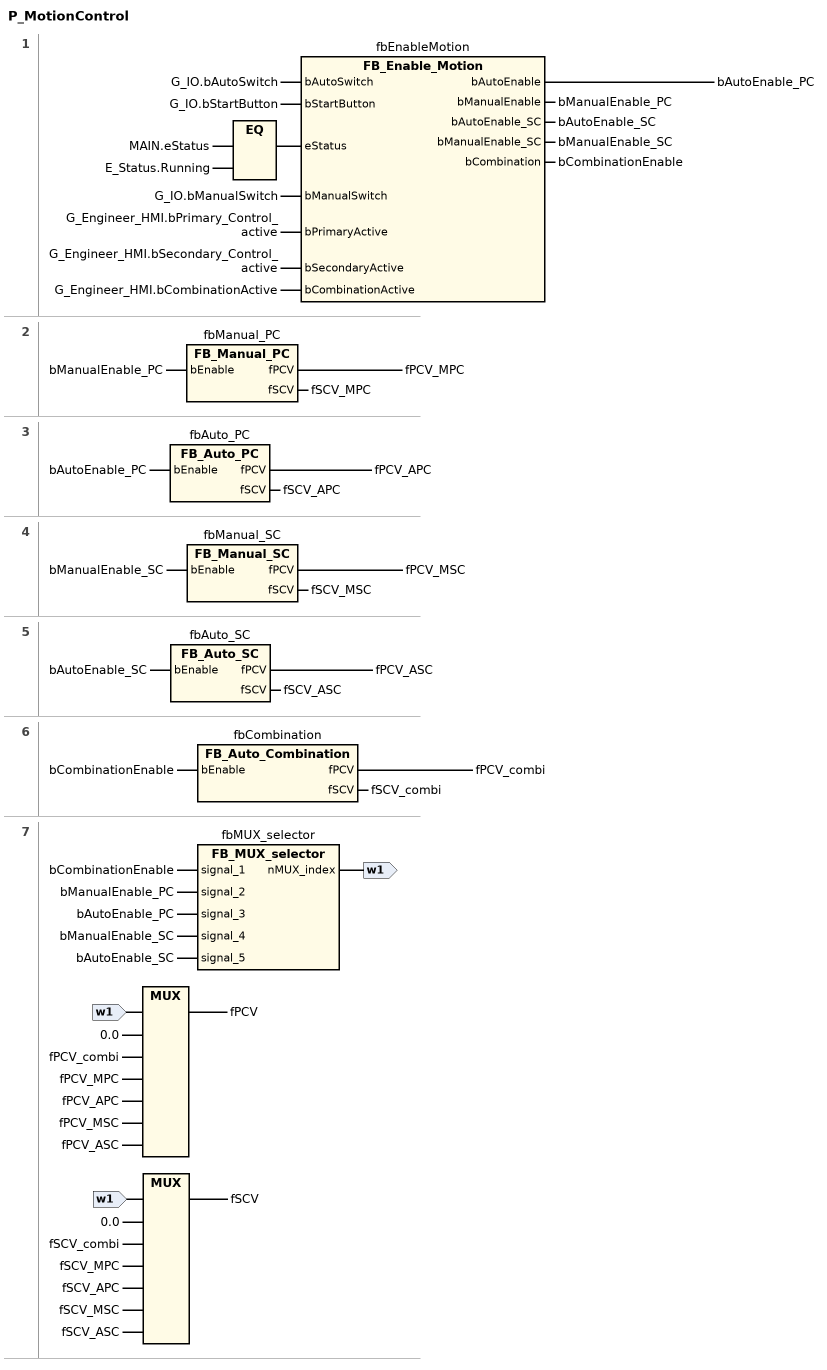
// NETWORK 1
fbEnableMotion(
    bAutoSwitch := G_IO.bAutoSwitch,
    bStartButton := G_IO.bStartButton,
    eStatus := MAIN.eStatus = E_Status.Running,
    bManualSwitch := G_IO.bManualSwitch,
    bPrimaryActive := G_Engineer_HMI.bPrimary_Control_active,
    bSecondaryActive := G_Engineer_HMI.bSecondary_Control_active,
    bCombinationActive := G_Engineer_HMI.bCombinationActive,
    bManualEnable => bManualEnable_PC,
    bAutoEnable_SC => bAutoEnable_SC,
    bManualEnable_SC => bManualEnable_SC,
    bCombination => bCombinationEnable); // FB_Enable_Motion
bAutoEnable_PC := fbEnableMotion.bAutoEnable;

// NETWORK 2
fbManual_PC(bEnable := bManualEnable_PC, fSCV => fSCV_MPC); // FB_Manual_PC
fPCV_MPC := fbManual_PC.fPCV;

// NETWORK 3
fbAuto_PC(bEnable := bAutoEnable_PC, fSCV => fSCV_APC); // FB_Auto_PC
fPCV_APC := fbAuto_PC.fPCV;

// NETWORK 4
fbManual_SC(bEnable := bManualEnable_SC, fSCV => fSCV_MSC); // FB_Manual_SC
fPCV_MSC := fbManual_SC.fPCV;

// NETWORK 5
fbAuto_SC(bEnable := bAutoEnable_SC, fSCV => fSCV_ASC); // FB_Auto_SC
fPCV_ASC := fbAuto_SC.fPCV;

// NETWORK 6
fbCombination(bEnable := bCombinationEnable, fSCV => fSCV_combi); // FB_Auto_Combination
fPCV_combi := fbCombination.fPCV;

// NETWORK 7
fbMUX_selector(
    signal_1 := bCombinationEnable,
    signal_2 := bManualEnable_PC,
    signal_3 := bAutoEnable_PC,
    signal_4 := bManualEnable_SC,
    signal_5 := bAutoEnable_SC); // FB_MUX_selector
fPCV := MUX(fbMUX_selector.nMUX_index, 0.0, fPCV_combi, fPCV_MPC, fPCV_APC, fPCV_MSC, fPCV_ASC);
fSCV := MUX(fbMUX_selector.nMUX_index, 0.0, fSCV_combi, fSCV_MPC, fSCV_APC, fSCV_MSC, fSCV_ASC);

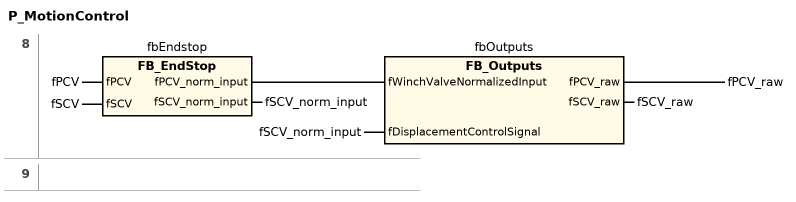
// NETWORK 8
fbEndstop(fPCV := fPCV, fSCV := fSCV, fSCV_norm_input => fSCV_norm_input); // FB_EndStop
fbOutputs(
    fWinchValveNormalizedInput := fbEndstop.fPCV_norm_input,
    fDisplacementControlSignal := fSCV_norm_input,
    fSCV_raw => fSCV_raw); // FB_Outputs
fPCV_raw := fbOutputs.fPCV_raw;

// NETWORK 9

END_PROGRAM

// ---- Function Blocks/FBs for Motion Control/FB_Enable_Motion.TcPOU
FUNCTION_BLOCK FB_Enable_Motion
VAR_INPUT
	bAutoSwitch								: BOOL;
	bStartButton							: BOOL;
	
	eStatus									: BOOL;
	
	bManualSwitch							: BOOL;
	
	bPrimaryActive							: BOOL;
	bSecondaryActive						: BOOL;
	bCombinationActive						: BOOL;
	
END_VAR
VAR_OUTPUT
	bAutoEnable 							: BOOL;
	bManualEnable 							: BOOL; 
	bAutoEnable_SC 							: BOOL; 
	bManualEnable_SC					    : BOOL;
	bCombination							: BOOL;
END_VAR
VAR
END_VAR

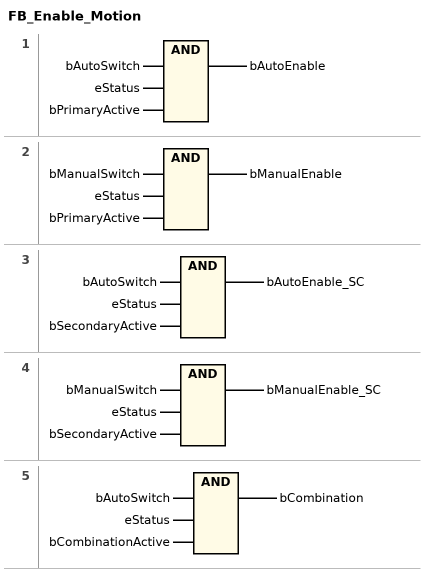
// NETWORK 1
bAutoEnable := bAutoSwitch AND eStatus AND bPrimaryActive;

// NETWORK 2
bManualEnable := bManualSwitch AND eStatus AND bPrimaryActive;

// NETWORK 3
bAutoEnable_SC := bAutoSwitch AND eStatus AND bSecondaryActive;

// NETWORK 4
bManualEnable_SC := bManualSwitch AND eStatus AND bSecondaryActive;

// NETWORK 5
bCombination := bAutoSwitch AND eStatus AND bCombinationActive;

END_FUNCTION_BLOCK

// ---- Function Blocks/FBs for Motion Control/FB_Manual_PC.TcPOU
FUNCTION_BLOCK FB_Manual_PC
VAR_INPUT
	bEnable					: BOOL;
END_VAR
VAR_OUTPUT
	fPCV					: LREAL;
	fSCV					: LREAL;
END_VAR
VAR
	//Function Blocks
	fbJoystick				: FB_Joystick;
	fbGetStartPos			: FB_StartPos;
	fbWinchVelIntegrator	: FB_Integrator;
	fbPID_Controller		: FB_PID_Controller;
	fbMUX_selector			: FB_MUX_selector;
	
	//Manual PosRef
	fWinchVelRefManual		: LREAL;
	fWInchVelRefAuto		: LREAL; //Brukes ikke
	fInitialWinchPos		: LREAL;
	
	//Valve signals
	fPCV_Manual			: LREAL;
	fPCV_PosRef			: LREAL;
	fPCV_Off			: LREAL;
	fSCV_On				: LREAL;
	fSCV_Off			: LREAL;
	
	
	//Notat på hva som skal til OPC UA
	//G_Motion_Control.fWinchPosRefManual
	


	END_VAR
VAR // added by the converter: edge detectors and wires of the graphical bodies
    _w1 : BOOL;
END_VAR

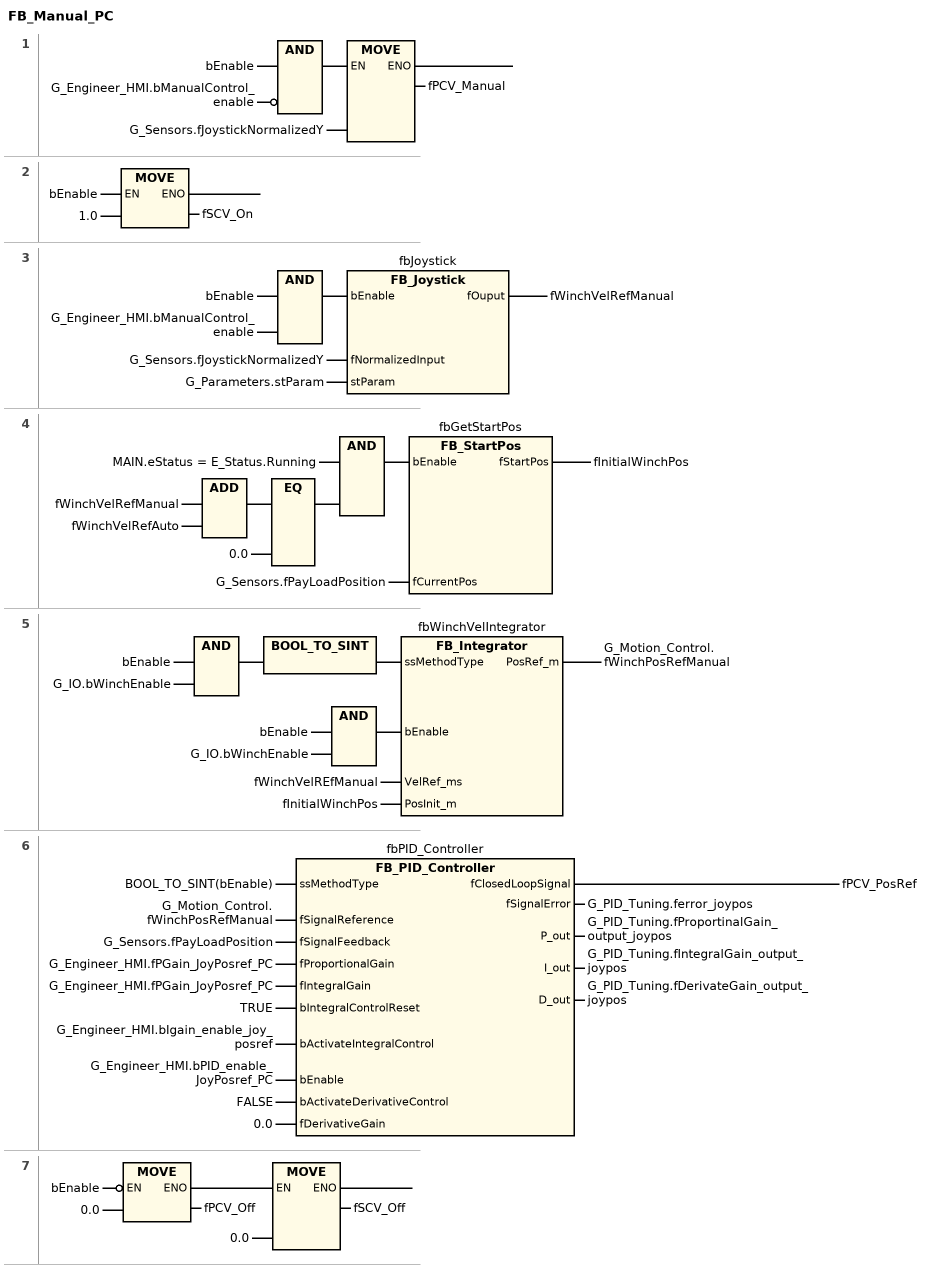
// NETWORK 1
IF bEnable AND NOT G_Engineer_HMI.bManualControl_enable THEN fPCV_Manual := G_Sensors.fJoystickNormalizedY; END_IF

// NETWORK 2
IF bEnable THEN fSCV_On := 1.0; END_IF

// NETWORK 3
fbJoystick(
    bEnable := bEnable AND G_Engineer_HMI.bManualControl_enable,
    fNormalizedInput := G_Sensors.fJoystickNormalizedY,
    stParam := G_Parameters.stParam); // FB_Joystick
fWinchVelRefManual := fbJoystick.fOuput;

// NETWORK 4
fbGetStartPos(bEnable := (MAIN.eStatus = E_Status.Running) AND fWinchVelRefManual + fWinchVelRefAuto = 0.0, fCurrentPos := G_Sensors.fPayLoadPosition); // FB_StartPos
fInitialWinchPos := fbGetStartPos.fStartPos;

// NETWORK 5
fbWinchVelIntegrator(
    ssMethodType := BOOL_TO_SINT(bEnable AND G_IO.bWinchEnable),
    bEnable := bEnable AND G_IO.bWinchEnable,
    VelRef_ms := fWinchVelREfManual,
    PosInit_m := fInitialWinchPos); // FB_Integrator
G_Motion_Control.fWinchPosRefManual := fbWinchVelIntegrator.PosRef_m;

// NETWORK 6
fbPID_Controller(
    ssMethodType := BOOL_TO_SINT(bEnable),
    fSignalReference := G_Motion_Control.fWinchPosRefManual,
    fSignalFeedback := G_Sensors.fPayLoadPosition,
    fProportionalGain := G_Engineer_HMI.fPGain_JoyPosref_PC,
    fIntegralGain := G_Engineer_HMI.fPGain_JoyPosref_PC,
    bIntegralControlReset := TRUE,
    bActivateIntegralControl := G_Engineer_HMI.bIgain_enable_joy_posref,
    bEnable := G_Engineer_HMI.bPID_enable_JoyPosref_PC,
    bActivateDerivativeControl := FALSE,
    fDerivativeGain := 0.0,
    fSignalError => G_PID_Tuning.ferror_joypos,
    P_out => G_PID_Tuning.fProportinalGain_output_joypos,
    I_out => G_PID_Tuning.fIntegralGain_output_joypos,
    D_out => G_PID_Tuning.fDerivateGain_output_joypos); // FB_PID_Controller
fPCV_PosRef := fbPID_Controller.fClosedLoopSignal;

// NETWORK 7
_w1 := NOT bEnable;
IF _w1 THEN fPCV_Off := 0.0; END_IF
IF _w1 THEN fSCV_Off := 0.0; END_IF

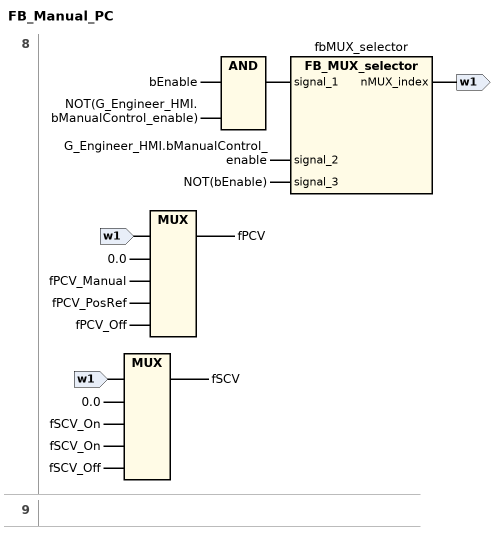
// NETWORK 8
fbMUX_selector(
    signal_1 := bEnable AND (NOT(G_Engineer_HMI.bManualControl_enable)),
    signal_2 := G_Engineer_HMI.bManualControl_enable,
    signal_3 := NOT(bEnable)); // FB_MUX_selector
fPCV := MUX(fbMUX_selector.nMUX_index, 0.0, fPCV_Manual, fPCV_PosRef, fPCV_Off);
fSCV := MUX(fbMUX_selector.nMUX_index, 0.0, fSCV_On, fSCV_On, fSCV_Off);

// NETWORK 9

END_FUNCTION_BLOCK

// ---- Function Blocks/FB_StartPos.TcPOU
FUNCTION_BLOCK FB_StartPos
VAR_INPUT
	bEnable 		: BOOL;
	fCurrentPos 	: LREAL;
END_VAR
VAR_OUTPUT
	fStartPos 		: LREAL;
END_VAR
VAR
END_VAR

IF bEnable THEN
	fStartPos := fStartPos;
	
ELSE 
	fStartPos := fCurrentPos;
END_IF

END_FUNCTION_BLOCK

// ---- Function Blocks/FB_Integrator.TcPOU
FUNCTION_BLOCK FB_Integrator
VAR_INPUT
	ssMethodType: SINT;
	bEnable: BOOL;
	VelRef_ms: LREAL;
	PosInit_m: LREAL;
END_VAR
VAR_OUTPUT
	PosRef_m: LREAL;
END_VAR
VAR
	c_DiscreteTimeIntegrator_IC: USINT;
	c_DiscreteTimeIntegrator_DS: LREAL;
END_VAR



CASE ssMethodType OF
    0: 
        (* SystemInitialize for Atomic SubSystem: '<Root>/FB_Integrator' *)
        (* InitializeConditions for DiscreteIntegrator: '<S1>/Discrete-Time Integrator' *)
        c_DiscreteTimeIntegrator_IC := 1;
        (* End of SystemInitialize for SubSystem: '<Root>/FB_Integrator' *)
    1: 
        (* Outputs for Atomic SubSystem: '<Root>/FB_Integrator' *)
        (* DiscreteIntegrator: '<S1>/Discrete-Time Integrator' *)

        IF c_DiscreteTimeIntegrator_IC <> 0 THEN 
            c_DiscreteTimeIntegrator_DS := PosInit_m;
        END_IF;

        (* Switch: '<S1>/Switch' *)

        IF bEnable THEN 
            (* Outport: '<Root>/PosRef_m' incorporates:
             *  DiscreteIntegrator: '<S1>/Discrete-Time Integrator' *)
            PosRef_m := c_DiscreteTimeIntegrator_DS;
        ELSE 
            (* Outport: '<Root>/PosRef_m' *)
            PosRef_m := PosInit_m;
        END_IF;

        (* End of Switch: '<S1>/Switch' *)
        

        (* Update for DiscreteIntegrator: '<S1>/Discrete-Time Integrator' *)
        c_DiscreteTimeIntegrator_IC := 0;
        c_DiscreteTimeIntegrator_DS := (0.01 * VelRef_ms) + c_DiscreteTimeIntegrator_DS;
        (* End of Outputs for SubSystem: '<Root>/FB_Integrator' *)
END_CASE;

END_FUNCTION_BLOCK

// ---- PIDs/FB_PID_Controller.TcPOU
FUNCTION_BLOCK FB_PID_Controller
VAR_INPUT
	ssMethodType: SINT;
	fSignalReference: LREAL;
	fSignalFeedback: LREAL;
	fProportionalGain: LREAL;
	fIntegralGain: LREAL;
	bIntegralControlReset: BOOL;
	bActivateIntegralControl: BOOL;
	bEnable: BOOL;
	bActivateDerivativeControl: BOOL;
	fDerivativeGain: LREAL;
END_VAR
VAR_OUTPUT
	fClosedLoopSignal: LREAL;
	fSignalError: LREAL;
	P_out: LREAL;
	I_out: LREAL;
	D_out: LREAL;
END_VAR
VAR
	rtb_Uk1: LREAL;
	rtb_Saturation: LREAL;
	rtb_TSamp: LREAL;
	c_DiscreteTimeIntegrator1_D: LREAL;
	UD_DSTATE: LREAL;
END_VAR



CASE ssMethodType OF
    0: 
        (* SystemInitialize for Atomic SubSystem: '<Root>/FB_PID_Controller' *)
        (* InitializeConditions for DiscreteIntegrator: '<S1>/Discrete-Time Integrator1' *)
        c_DiscreteTimeIntegrator1_D := 0.0;
        (* InitializeConditions for UnitDelay: '<S2>/UD'
         *
         * Block description for '<S2>/UD':
         *  
         *  Store in Global RAM *)
        UD_DSTATE := 0.0;
        (* End of SystemInitialize for SubSystem: '<Root>/FB_PID_Controller' *)
    1: 
        (* Outputs for Atomic SubSystem: '<Root>/FB_PID_Controller' *)
        (* Sum: '<S1>/Sum' *)
        fSignalError := fSignalReference - fSignalFeedback;
        (* Product: '<S1>/Product' *)
        P_out := fProportionalGain * fSignalError;
        (* DiscreteIntegrator: '<S1>/Discrete-Time Integrator1' *)

        IF bIntegralControlReset THEN 
            c_DiscreteTimeIntegrator1_D := 0.0;
        END_IF;

        (* Switch: '<S1>/Switch2' incorporates:
         *  Constant: '<S1>/Constant'
         *  DiscreteIntegrator: '<S1>/Discrete-Time Integrator1' *)

        IF bActivateIntegralControl THEN 
            I_out := c_DiscreteTimeIntegrator1_D;
        ELSE 
            I_out := 0.0;
        END_IF;

        (* End of Switch: '<S1>/Switch2' *)
        

        (* Sum: '<S1>/Sum5' *)
        rtb_Uk1 := P_out + I_out;
        (* Saturate: '<S1>/Saturation' *)

        IF rtb_Uk1 > 1.0 THEN 
            rtb_Saturation := 1.0;
        ELSIF rtb_Uk1 >= -1.0 THEN 
            rtb_Saturation := rtb_Uk1;
        ELSE 
            rtb_Saturation := -1.0;
        END_IF;

        (* End of Saturate: '<S1>/Saturation' *)
        

        (* SampleTimeMath: '<S2>/TSamp' incorporates:
         *  Product: '<S1>/Product2'
         *
         * About '<S2>/TSamp':
         *  y = u * K where K = 1 / ( w * Ts )
         *   *)
        rtb_TSamp := (fSignalError * fDerivativeGain) * 100.0;
        (* Switch: '<S1>/Switch3' incorporates:
         *  Constant: '<S1>/Constant2'
         *  Sum: '<S2>/Diff'
         *  UnitDelay: '<S2>/UD'
         *
         * Block description for '<S2>/Diff':
         *  
         *  Add in CPU
         *
         * Block description for '<S2>/UD':
         *  
         *  Store in Global RAM *)

        IF bActivateDerivativeControl THEN 
            D_out := rtb_TSamp - UD_DSTATE;
        ELSE 
            D_out := 0.0;
        END_IF;

        (* End of Switch: '<S1>/Switch3' *)
        

        (* Switch: '<S1>/Switch1' *)

        IF bEnable THEN 
            (* Sum: '<S1>/Sum2' *)
            fClosedLoopSignal := rtb_Saturation + D_out;
            (* Saturate: '<S1>/Saturation1' *)

            IF fClosedLoopSignal > 1.0 THEN 
                (* Outport: '<Root>/fClosedLoopSignal' *)
                fClosedLoopSignal := 1.0;
            ELSIF fClosedLoopSignal < -1.0 THEN 
                (* Outport: '<Root>/fClosedLoopSignal' *)
                fClosedLoopSignal := -1.0;
            END_IF;

            (* End of Saturate: '<S1>/Saturation1' *)
        ELSE 
            (* Outport: '<Root>/fClosedLoopSignal' incorporates:
             *  Constant: '<S1>/Constant1' *)
            fClosedLoopSignal := 0.0;
        END_IF;

        (* End of Switch: '<S1>/Switch1' *)
        

        (* Update for DiscreteIntegrator: '<S1>/Discrete-Time Integrator1' incorporates:
         *  Product: '<S1>/Divide'
         *  Product: '<S1>/Product1'
         *  Sum: '<S1>/Sum1'
         *  Sum: '<S1>/Sum3' *)
        c_DiscreteTimeIntegrator1_D := (((((rtb_Saturation - rtb_Uk1) / fProportionalGain) + fSignalError) * fIntegralGain) * 0.01) + c_DiscreteTimeIntegrator1_D;

        IF c_DiscreteTimeIntegrator1_D > 1.0 THEN 
            c_DiscreteTimeIntegrator1_D := 1.0;
        ELSIF c_DiscreteTimeIntegrator1_D < -1.0 THEN 
            c_DiscreteTimeIntegrator1_D := -1.0;
        END_IF;

        (* End of Update for DiscreteIntegrator: '<S1>/Discrete-Time Integrator1' *)
        

        (* Update for UnitDelay: '<S2>/UD'
         *
         * Block description for '<S2>/UD':
         *  
         *  Store in Global RAM *)
        UD_DSTATE := rtb_TSamp;
        (* End of Outputs for SubSystem: '<Root>/FB_PID_Controller' *)
END_CASE;

END_FUNCTION_BLOCK

// ---- Function Blocks/FBs for Motion Control/FB_MUX_selector.TcPOU
FUNCTION_BLOCK FB_MUX_selector
VAR_INPUT
	//signal_0								: BOOL; //SLik det er nå blir utgangen 0 om ingen er valgt
	signal_1		 						: BOOL; 
	signal_2 								: BOOL;
	signal_3							    : BOOL;
	signal_4	 							: BOOL; 
	signal_5								: BOOL;
END_VAR
VAR_OUTPUT
nMUX_index								: INT;
END_VAR
VAR	
END_VAR

IF signal_1 THEN
	nMUX_index := 1;
ELSIF signal_2 THEN
	nMUX_index := 2;
ELSIF signal_3 THEN
	nMUX_index := 3;
ELSIF signal_4 THEN
	nMUX_index := 4;
ELSIF signal_5 THEN
	nMUX_index := 5;
ELSE
	nMUX_index := 0;	
END_IF

END_FUNCTION_BLOCK

// ---- Function Blocks/FBs for Motion Control/FB_Auto_PC.TcPOU
FUNCTION_BLOCK FB_Auto_PC
VAR_INPUT
	bEnable				: BOOL;
END_VAR	
VAR_OUTPUT
	fPCV				: LREAL;
	fSCV				: LREAL;

END_VAR
VAR
	//Valvesignals
fPCV_startpos				: LREAL;
fPCV_sine					: LREAL;
fPCV_Off					: LREAL;

fSCV_On						: LREAL;
fSCV_Off					: LREAL;

	//Function Blocks
	fbAutoStartPos		: FB_AutoStartPos;
	fbAutoSineMotion	: FB_AutoSineMotion;
	
	fbClock				: FB_Clock;
	fbMUX_selector		: FB_MUX_selector;
	
	
	bStartPosOK			: BOOL;

END_VAR
VAR // added by the converter: edge detectors and wires of the graphical bodies
    _w1 : LREAL;
    _w2 : BOOL;
END_VAR

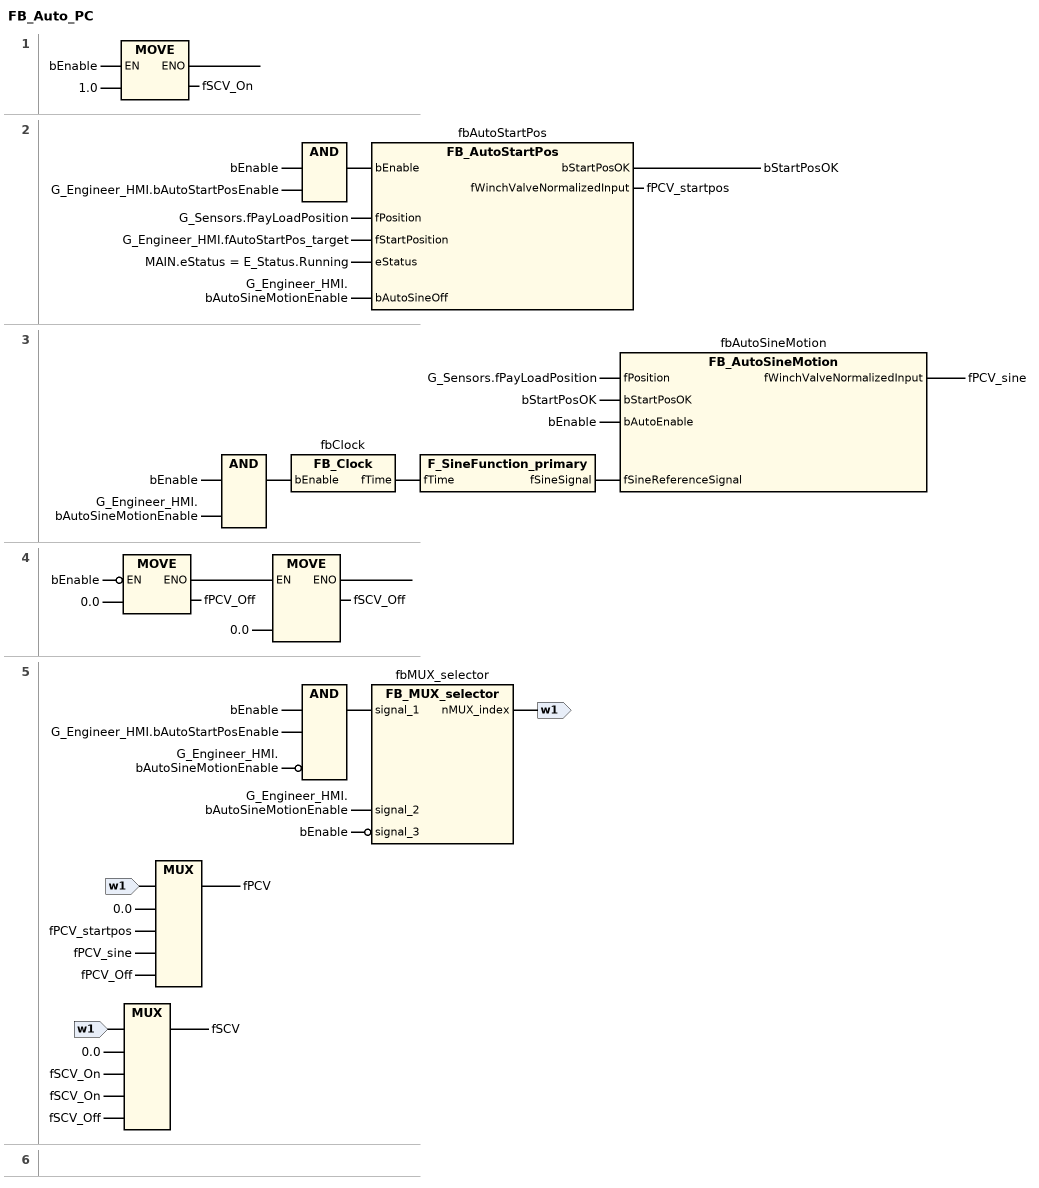
// NETWORK 1
IF bEnable THEN fSCV_On := 1.0; END_IF

// NETWORK 2
fbAutoStartPos(
    bEnable := bEnable AND G_Engineer_HMI.bAutoStartPosEnable,
    fPosition := G_Sensors.fPayLoadPosition,
    fStartPosition := G_Engineer_HMI.fAutoStartPos_target,
    eStatus := MAIN.eStatus = E_Status.Running,
    bAutoSineOff := G_Engineer_HMI.bAutoSineMotionEnable,
    fWinchValveNormalizedInput => fPCV_startpos); // FB_AutoStartPos
bStartPosOK := fbAutoStartPos.bStartPosOK;

// NETWORK 3
fbClock(bEnable := bEnable AND G_Engineer_HMI.bAutoSineMotionEnable); // FB_Clock
F_SineFunction_primary(fTime := fbClock.fTime, fSineSignal => _w1);
fbAutoSineMotion(
    fPosition := G_Sensors.fPayLoadPosition,
    bStartPosOK := bStartPosOK,
    bAutoEnable := bEnable,
    fSineReferenceSignal := _w1); // FB_AutoSineMotion
fPCV_sine := fbAutoSineMotion.fWinchValveNormalizedInput;

// NETWORK 4
_w2 := NOT bEnable;
IF _w2 THEN fPCV_Off := 0.0; END_IF
IF _w2 THEN fSCV_Off := 0.0; END_IF

// NETWORK 5
fbMUX_selector(
    signal_1 := bEnable AND G_Engineer_HMI.bAutoStartPosEnable AND NOT G_Engineer_HMI.bAutoSineMotionEnable,
    signal_2 := G_Engineer_HMI.bAutoSineMotionEnable,
    signal_3 := NOT bEnable); // FB_MUX_selector
fPCV := MUX(fbMUX_selector.nMUX_index, 0.0, fPCV_startpos, fPCV_sine, fPCV_Off);
fSCV := MUX(fbMUX_selector.nMUX_index, 0.0, fSCV_On, fSCV_On, fSCV_Off);

// NETWORK 6

END_FUNCTION_BLOCK

// ---- Function Blocks/FBs Auto Control/FB_AutoStartPos.TcPOU
FUNCTION_BLOCK FB_AutoStartPos
VAR_INPUT
	bEnable 						: BOOL; 
	fPosition						: LREAL;
	fStartPosition					: LREAL;
	
	eStatus 						: BOOL; //E_Status;
	bAutoSineOff					: BOOL;
END_VAR
VAR_OUTPUT
	bStartPosOK						: BOOL;
	fWinchValveNormalizedInput 		: LREAL;
END_VAR


VAR
	fbPID							: FB_PID_Controller;
	fPosition_error					: LREAL;
	fProportinalGain_output			: LREAL;
	fIntegralGain_output			: LREAL;
	fDerivateGain_output			: LREAL;
	bEnableValveOutputWinch			: BOOL;	
	
	//Soft Start
	u								: LREAL;
	y								: LREAL;
	fTotal_distance					: LREAL;
	bAutoSineOff_prev				: BOOL;
END_VAR

IF bEnable  THEN

/////Soft Start//////

(*
IF NOT(bAutoSineOff) AND bAutoSineOff_prev THEN
fTotal_distance := ABS(fStartPosition - fPosition);
END_IF

bAutoSineOff_prev := bAutoSineOff;

u := fPosition_error/fTotal_distance;

IF u > 0.5 THEN
y := 1 - ((3*u*u) - (2*u*u*u)); 
END_IF

IF u < 0.5 THEN
	y := ((3*u*u) - (2*u*u*u)); 
END_IF

IF u < 0.0 THEN
	u := 0.0;
END_IF*)


		
fbPID(
	ssMethodType := BOOL_TO_SINT(bEnable),
	fSignalReference := fStartPosition,
	fSignalFeedback := fPosition,
	fProportionalGain := G_Engineer_HMI.fPgain_MOOG,
	fIntegralGain := G_Engineer_HMI.fIgain_MOOG,
	bActivateIntegralControl := G_Engineer_HMI.bIenable_MOOG,
	bEnable := TRUE,
	bActivateDerivativeControl := FALSE,
	fDerivativeGain := 0.0,
	fClosedLoopSignal => fWinchValveNormalizedInput,
	fSignalError => G_Motion_Control.fPosition_error_StartPos,
	P_out => G_PID_Tuning.fProportinalGain_output_MOOG,
	I_out => G_PID_Tuning.fIntegralGain_output_MOOG,
	D_out => G_PID_Tuning.fDerivateGain_output_MOOG
	);
	
	
	//Make output global for plot	
	G_PID_Tuning.PID_output_MOOG := fWinchValveNormalizedInput;

	
IF ABS(G_Motion_Control.fPosition_error_StartPos) < 0.05 THEN //Tidligere denne: fPosition_error i ABS
		bStartPosOK := TRUE;
END_IF
		
ELSE
	bStartPosOK := FALSE;
END_IF

END_FUNCTION_BLOCK

// ---- Function Blocks/FBs Auto Control/FB_AutoSineMotion.TcPOU
FUNCTION_BLOCK FB_AutoSineMotion
VAR_INPUT 
	fPosition : LREAL; 
	bStartPosOK						: BOOL;
	bAutoEnable : BOOL; 
	// eStatus : BOOL;
    fSineReferenceSignal                  : LREAL; 
END_VAR


VAR_OUTPUT
	fWinchValveNormalizedInput 		: LREAL;
END_VAR
VAR
	bEnable : BOOL; // Forblir TRUE bnår og etter bStartPosOk er TRUE?
	fbPID						:FB_PID_Controller;
	fPosition_error					: LREAL;
	fProportinalGain_output			: LREAL;
	fIntegralGain_output			: LREAL;
	fDerivateGain_output			: LREAL;
	bEnableValveOutputWinch			: BOOL;	 
END_VAR

IF NOT(G_IO.bStartButton) THEN //Tidligere var denne koblet til bAutoEnable
	bEnable := FALSE;
	G_Engineer_HMI.bAutoSineMotionEnable := FALSE;
	fWinchValveNormalizedInput := 0.0;
ELSIF bStartPosOK AND bAutoEnable THEN
	bEnable := TRUE;
END_IF

IF bEnable THEN	
	
G_Motion_Control.fSineReferenceSignal := fSineReferenceSignal;
	
	

		
		fbPID(
	ssMethodType := BOOL_TO_SINT(bEnable),
	fSignalReference := fSineReferenceSignal,
	fSignalFeedback := fPosition,
	fProportionalGain := G_Engineer_HMI.fPGain_MOOG,
	fIntegralGain :=  G_Engineer_HMI.fIGain_MOOG,
	bActivateIntegralControl := G_Engineer_HMI.bIenable_MOOG,
	bEnable := TRUE,
	bActivateDerivativeControl := FALSE,
	fDerivativeGain := 0.0,
	fClosedLoopSignal => fWinchValveNormalizedInput,
	fSignalError =>G_Motion_Control.fPosition_error_SineMotion,
	P_out => G_PID_Tuning.fProportinalGain_output_MOOG,
	I_out => G_PID_Tuning.fIntegralGain_output_MOOG,
	D_out => G_PID_Tuning.fDerivateGain_output_MOOG
	);
		
		
	
	//Make output global for plot		
		G_PID_Tuning.PID_output_MOOG := fWinchValveNormalizedInput;
		


END_IF

END_FUNCTION_BLOCK

// ---- Function Blocks/FB_Clock.TcPOU
FUNCTION_BLOCK FB_Clock
VAR_INPUT
	bEnable : BOOL;
END_VAR
VAR_OUTPUT
	fTime : LREAL;
END_VAR
VAR
	stParameter : ST_Parameters;
END_VAR

IF bEnable THEN
	fTime := fTime + stParameter.fCyclicTime;
ELSE
	fTime := 0.0; 	
END_IF

END_FUNCTION_BLOCK

// ---- Functions/F_SineFunction_primary.TcPOU
FUNCTION F_SineFunction_primary : LREAL
VAR_INPUT
	fTime 				: LREAL;
END_VAR
VAR_OUTPUT
	fSineSignal 		: LREAL;
END_VAR
VAR
	u					: LREAL;
	ft_ENV				: LREAL;
	y					: LREAL;
	
END_VAR

ft_ENV := G_Engineer_HMI.ft_ENV;

u := fTime/ft_ENV;

IF u > 1.0 THEN
	u := 1.0;
END_IF

y := (3.0*u*u) - (2.0*u*u*u);

fSineSignal := y* G_Engineer_HMI.fAmp * SIN(2.0 * PI * G_Engineer_HMI.fFreq * fTime) + G_Engineer_HMI.fSinemidpoint;

END_FUNCTION

// ---- Function Blocks/FBs for Motion Control/FB_Manual_SC.TcPOU
FUNCTION_BLOCK FB_Manual_SC
VAR_INPUT
	bEnable			: BOOL;
	
END_VAR
VAR_OUTPUT
	fPCV				: LREAL;
	fSCV				: LREAL;
END_VAR
VAR
//Set fPCV
fPCV_set				: LREAL := 1.0;



//Function Blocks
fbDisplacementControl		: FB_DisplacementControl; //slik det er nå må Manuel SC være på for å endre dis, 
													  //kan endres til bare running og knappen

fbJoystick					: FB_Joystick;
fbGetStartPos				: FB_StartPos;
fbWinchVelIntegrator		: FB_Integrator;
fbPID_OL					: FB_PID_Controller;
fbDeadband					: FB_Deadband;
fbDisplacementControl_SC	: FB_DisplacementControl_SC;

fbMUX_selector				: FB_MUX_selector;

fbTarget_dis				: FB_Target_displacement;
fbGain_Chooser_P			: FB_GainChooser;
fbGain_Chooser_I			: FB_GainChooser;
fb_ControlReset				: FB_ControlReset_SC;


//Variables
fWinchVelRefManual			: LREAL;
fWinchVelRefAuto			: LREAL;
fInitialWinchPos			: LREAL;

//Deaband
fDeadbandComp_out			: LREAL;

//Outer Loop output
fSC_ClosedLoopSingal		: LREAL;

//Valve signals
fSCV_target					: LREAL;
fSCV_Posref					: LREAL;
fSCV_Off					: LREAL;

fPCV_On						: LREAL;
fPCV_Off					: LREAL;

//FeedForward
fbFeedforward				: FB_Feedforward_SC;
fbDerivator					: FB_Derivator;
fAlpha						: LREAL;
fKff						: LREAL := 1.0;



END_VAR
VAR // added by the converter: edge detectors and wires of the graphical bodies
    _w1 : BOOL;
END_VAR

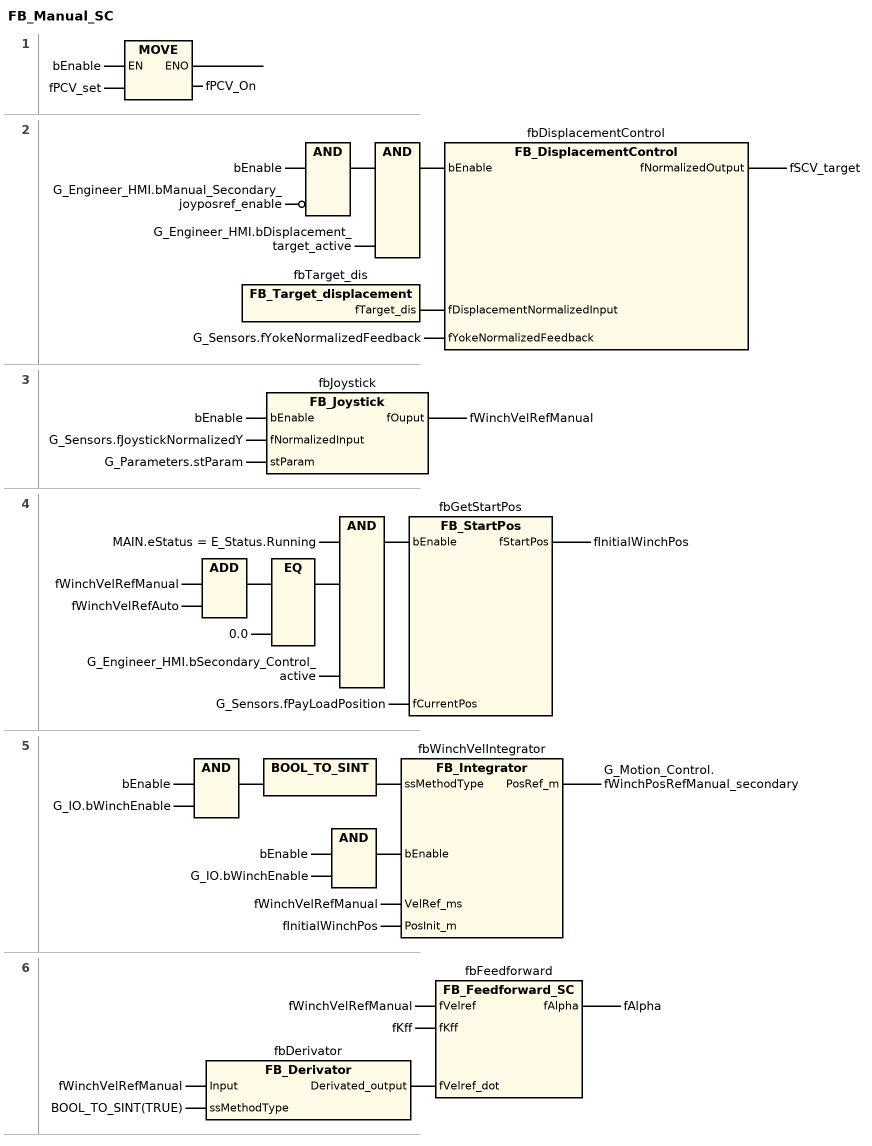
// NETWORK 1
IF bEnable THEN fPCV_On := fPCV_set; END_IF

// NETWORK 2
fbTarget_dis(); // FB_Target_displacement
fbDisplacementControl(
    bEnable := (bEnable AND NOT G_Engineer_HMI.bManual_Secondary_joyposref_enable) AND G_Engineer_HMI.bDisplacement_target_active,
    fDisplacementNormalizedInput := fbTarget_dis.fTarget_dis,
    fYokeNormalizedFeedback := G_Sensors.fYokeNormalizedFeedback); // FB_DisplacementControl
fSCV_target := fbDisplacementControl.fNormalizedOutput;

// NETWORK 3
fbJoystick(
    bEnable := bEnable,
    fNormalizedInput := G_Sensors.fJoystickNormalizedY,
    stParam := G_Parameters.stParam); // FB_Joystick
fWinchVelRefManual := fbJoystick.fOuput;

// NETWORK 4
fbGetStartPos(bEnable := (MAIN.eStatus = E_Status.Running) AND fWinchVelRefManual + fWinchVelRefAuto = 0.0 AND G_Engineer_HMI.bSecondary_Control_active, fCurrentPos := G_Sensors.fPayLoadPosition); // FB_StartPos
fInitialWinchPos := fbGetStartPos.fStartPos;

// NETWORK 5
fbWinchVelIntegrator(
    ssMethodType := BOOL_TO_SINT(bEnable AND G_IO.bWinchEnable),
    bEnable := bEnable AND G_IO.bWinchEnable,
    VelRef_ms := fWinchVelRefManual,
    PosInit_m := fInitialWinchPos); // FB_Integrator
G_Motion_Control.fWinchPosRefManual_secondary := fbWinchVelIntegrator.PosRef_m;

// NETWORK 6
fbDerivator(Input := fWinchVelRefManual, ssMethodType := BOOL_TO_SINT(TRUE)); // FB_Derivator
fbFeedforward(fVelref := fWinchVelRefManual, fKff := fKff, fVelref_dot := fbDerivator.Derivated_output); // FB_Feedforward_SC
fAlpha := fbFeedforward.fAlpha;

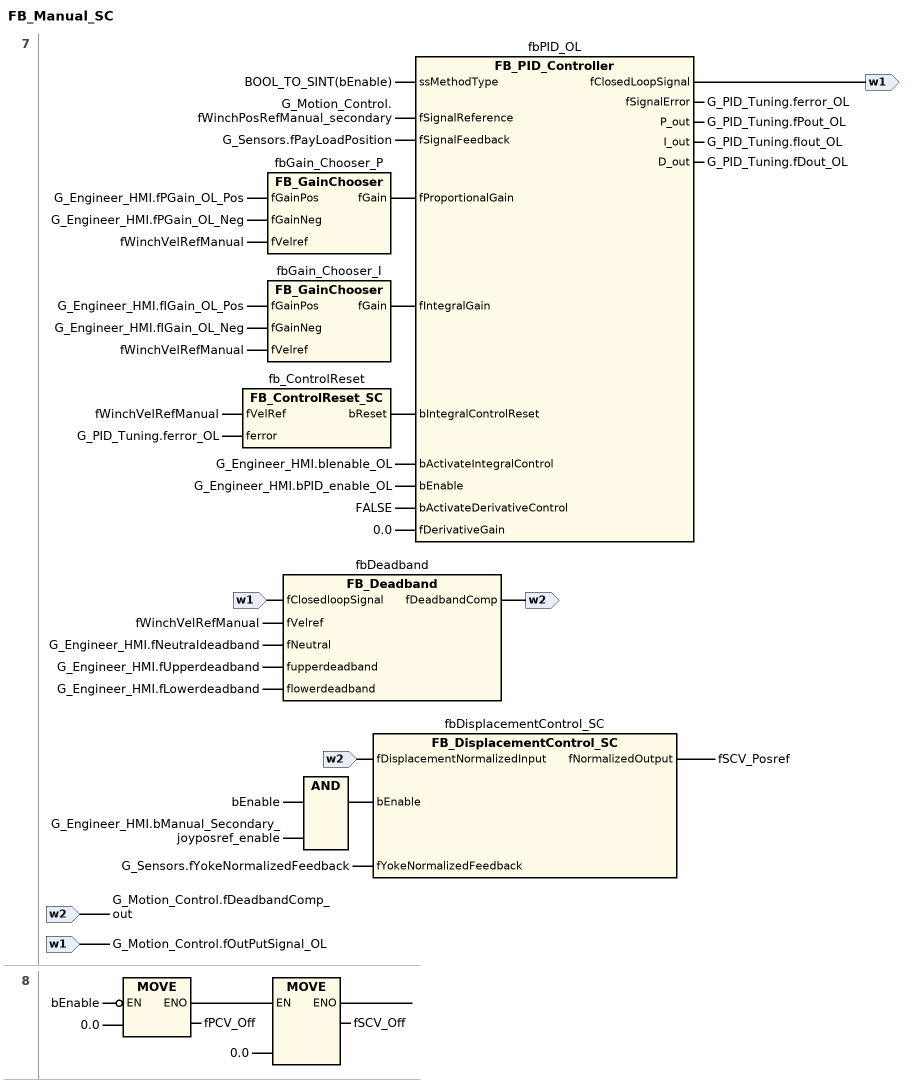
// NETWORK 7
fbGain_Chooser_P(
    fGainPos := G_Engineer_HMI.fPGain_OL_Pos,
    fGainNeg := G_Engineer_HMI.fPGain_OL_Neg,
    fVelref := fWinchVelRefManual); // FB_GainChooser
fbGain_Chooser_I(
    fGainPos := G_Engineer_HMI.fIGain_OL_Pos,
    fGainNeg := G_Engineer_HMI.fIGain_OL_Neg,
    fVelref := fWinchVelRefManual); // FB_GainChooser
fb_ControlReset(fVelRef := fWinchVelRefManual, ferror := G_PID_Tuning.ferror_OL); // FB_ControlReset_SC
fbPID_OL(
    ssMethodType := BOOL_TO_SINT(bEnable),
    fSignalReference := G_Motion_Control.fWinchPosRefManual_secondary,
    fSignalFeedback := G_Sensors.fPayLoadPosition,
    fProportionalGain := fbGain_Chooser_P.fGain,
    fIntegralGain := fbGain_Chooser_I.fGain,
    bIntegralControlReset := fb_ControlReset.bReset,
    bActivateIntegralControl := G_Engineer_HMI.bIenable_OL,
    bEnable := G_Engineer_HMI.bPID_enable_OL,
    bActivateDerivativeControl := FALSE,
    fDerivativeGain := 0.0,
    fSignalError => G_PID_Tuning.ferror_OL,
    P_out => G_PID_Tuning.fPout_OL,
    I_out => G_PID_Tuning.fIout_OL,
    D_out => G_PID_Tuning.fDout_OL); // FB_PID_Controller
fbDeadband(
    fClosedloopSignal := fbPID_OL.fClosedLoopSignal,
    fVelref := fWinchVelRefManual,
    fNeutral := G_Engineer_HMI.fNeutraldeadband,
    fupperdeadband := G_Engineer_HMI.fUpperdeadband,
    flowerdeadband := G_Engineer_HMI.fLowerdeadband); // FB_Deadband
fbDisplacementControl_SC(
    fDisplacementNormalizedInput := fbDeadband.fDeadbandComp,
    bEnable := bEnable AND G_Engineer_HMI.bManual_Secondary_joyposref_enable,
    fYokeNormalizedFeedback := G_Sensors.fYokeNormalizedFeedback); // FB_DisplacementControl_SC
fSCV_Posref := fbDisplacementControl_SC.fNormalizedOutput;
G_Motion_Control.fDeadbandComp_out := fbDeadband.fDeadbandComp;
G_Motion_Control.fOutPutSignal_OL := fbPID_OL.fClosedLoopSignal;

// NETWORK 8
_w1 := NOT bEnable;
IF _w1 THEN fPCV_Off := 0.0; END_IF
IF _w1 THEN fSCV_Off := 0.0; END_IF

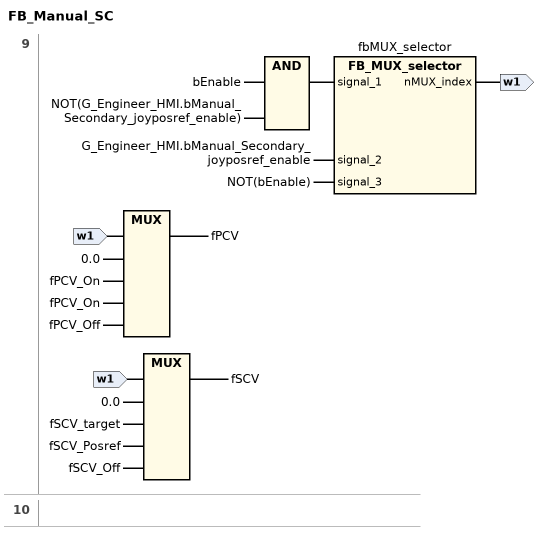
// NETWORK 9
fbMUX_selector(
    signal_1 := bEnable AND (NOT(G_Engineer_HMI.bManual_Secondary_joyposref_enable)),
    signal_2 := G_Engineer_HMI.bManual_Secondary_joyposref_enable,
    signal_3 := NOT(bEnable)); // FB_MUX_selector
fPCV := MUX(fbMUX_selector.nMUX_index, 0.0, fPCV_On, fPCV_On, fPCV_Off);
fSCV := MUX(fbMUX_selector.nMUX_index, 0.0, fSCV_target, fSCV_Posref, fSCV_Off);

// NETWORK 10

END_FUNCTION_BLOCK

// ---- Function Blocks/FB_DisplacementControl.TcPOU
FUNCTION_BLOCK FB_DisplacementControl 
VAR_INPUT
	bEnable 						: BOOL; 
	
	fDisplacementNormalizedInput 	: LREAL; 
	fYokeNormalizedFeedback 		: LREAL; 
	
	fVelRef							: LREAL;
END_VAR
VAR_OUTPUT
	fNormalizedOutput 				: LREAL; 
END_VAR

VAR PERSISTENT
	fProportionalGain 				: LREAL := 1.0;
	fIntegralGain					: LREAL;
	fDerivateGain					: LREAL;
END_VAR

VAR
	fbPID_Conroller					: FB_PID_Controller;
	fbResetInt						: FB_ResetIntegralController;
	bResetInt						: BOOL;
	
	fYoke_error						: LREAL;
	fProportinalGain_output			: LREAL;
	fIntegralGain_output			: LREAL;
	fDerivateGain_output			: LREAL;
END_VAR

IF bEnable THEN
	
	IF G_PID_Tuning.fYoke_error > 0.0 THEN //Kan legge inn en velref  istedet for feilen
	fProportionalGain := G_Engineer_HMI.fPGain_IL_Pos;
	fIntegralGain := G_Engineer_HMI.fIGain_IL_Pos;
	fDerivateGain := G_Engineer_HMI.fDGain_IL_Pos;
ELSIF G_PID_Tuning.fYoke_error < 0.0 THEN
	fProportionalGain := G_Engineer_HMI.fPGain_IL_Neg;
	fIntegralGain := G_Engineer_HMI.fIGain_IL_Neg;
	fDerivateGain := G_Engineer_HMI.fDGain_IL_Neg;
ELSE
	fProportionalGain := G_Engineer_HMI.fPGain_IL_Pos;
	fIntegralGain := G_Engineer_HMI.fIGain_IL_Pos;
	fDerivateGain := G_Engineer_HMI.fDGain_IL_Pos;
END_IF
	

		
		fbPID_Conroller(
	ssMethodType := BOOL_TO_SINT(bEnable),
	fSignalReference := fDisplacementNormalizedInput,
	fSignalFeedback := fYokeNormalizedFeedback,
	fProportionalGain := fProportionalGain,
	fIntegralGain := fIntegralGain,
	bActivateIntegralControl := G_Engineer_HMI.bIenable_IL,
	bEnable := bEnable,
	bIntegralControlReset := NOT(bEnable),
	bActivateDerivativeControl := G_Engineer_HMI.bDenable_IL,
	fDerivativeGain := fDerivateGain,
	fClosedLoopSignal => fNormalizedOutput,
	fSignalError =>G_PID_Tuning.fYoke_error,
	P_out => G_PID_Tuning.fPout_IL,
	I_out => G_PID_Tuning.fIout_IL,
	D_out => G_PID_Tuning.fDout_IL
	);	
	
(*fbResetInt(
	fVRef := 0.0,
	fErrorMax := G_Engineer_HMI.fMaxerror_dis,
	fError := G_PID_Tuning.fYoke_error,
	bReset => bResetInt
	);*)
	
	//Make Output global for plot
	G_PID_Tuning.PID_output_IL := fNormalizedOutput;
	
ELSE 
	fNormalizedOutput := 0.0; // Ingen output uten aktivering
END_IF

END_FUNCTION_BLOCK

// ---- PIDs/FB_ResetIntegralController.TcPOU
FUNCTION_BLOCK FB_ResetIntegralController
VAR_INPUT
	fVRef: LREAL;
	fErrorMax: LREAL;
	fError: LREAL;
END_VAR
VAR_OUTPUT
	bReset: BOOL;
END_VAR
VAR
	rtb_Reset: DINT;
END_VAR


(* Outputs for Atomic SubSystem: '<Root>/FB_ResetIntegralController' *)
(* MATLAB Function: '<S1>/MATLAB Function' *)
(* MATLAB Function 'FB_ResetIntegralController/MATLAB Function': '<S2>:1' *)
(* '<S2>:1:3' if abs(vRef) > 0 || abs(error) > errorMax *)

IF ABS(fVRef) > 0.0 THEN 
    (* '<S2>:1:4' Reset = 0; *)
    rtb_Reset := 0;
ELSIF ABS(fError) > fErrorMax THEN //////I simulink er det ABS(fError) > fErrorMax
    (* '<S2>:1:4' Reset = 0; *)
    rtb_Reset := 0;
ELSE 
    (* '<S2>:1:5' else *)
    (* '<S2>:1:6' Reset = 1; *)
    rtb_Reset := 1;
END_IF;

(* End of MATLAB Function: '<S1>/MATLAB Function' *)


(* Outport: '<Root>/bReset' incorporates:
 *  DataTypeConversion: '<S1>/Data Type Conversion' *)
bReset := rtb_Reset <> 0;
(* End of Outputs for SubSystem: '<Root>/FB_ResetIntegralController' *)

END_FUNCTION_BLOCK

// ---- Function Blocks/Deadband Comp/FB_Deadband.TcPOU
FUNCTION_BLOCK FB_Deadband
VAR_INPUT
	fClosedloopSignal	: LREAL;
	fVelref				: LREAL;
	fNeutral			: LREAL;
	fupperdeadband		: LREAL;
	flowerdeadband		: LREAL;
	
END_VAR
VAR_OUTPUT
	fDeadbandComp		: LREAL;
END_VAR
VAR
END_VAR



IF fVelref > 0.0 THEN
	fDeadbandComp := LIMIT(fNeutral,fupperdeadband + fClosedloopSignal,1.0);
ELSIF fVelref < 0.0 THEN
	fDeadbandComp := LIMIT(0.0,flowerdeadband + fClosedloopSignal,fNeutral); //Kanskje minus her men tror input blir - så da blir det fikset
ELSE
	fDeadbandComp := LIMIT(0.1,fNeutral + fClosedloopSignal,1.0);
END_IF

END_FUNCTION_BLOCK

// ---- Function Blocks/FB_DisplacementControl_SC.TcPOU
FUNCTION_BLOCK FB_DisplacementControl_SC 
VAR_INPUT
	
	fDisplacementNormalizedInput 	: LREAL;
	bEnable 						: BOOL; 
	fYokeNormalizedFeedback 		: LREAL;
	
	fVelRef							: LREAL;
	
END_VAR
VAR_OUTPUT
	fNormalizedOutput 				: LREAL; 
END_VAR

VAR PERSISTENT
	
END_VAR

VAR
	fProportionalGain 				: LREAL;
	fIntegralGain					: LREAL;
	fDerivateGain					: LREAL;	


	fbPID_IL						: FB_PID_Controller;
	fbPID_new						: FB_PID_Controller;
	fYoke_error						: LREAL;
	fProportinalGain_output			: LREAL;
	fIntegralGain_output			: LREAL;
	fDerivateGain_output			: LREAL;
END_VAR


IF bEnable THEN
	


IF fVelRef > 0.0 THEN
	fProportionalGain := G_Engineer_HMI.fPGain_IL_Pos;
	fIntegralGain := G_Engineer_HMI.fIGain_IL_Pos;
	fDerivateGain := G_Engineer_HMI.fDGain_IL_Pos;
ELSIF fVelRef < 0.0 THEN
	fProportionalGain := G_Engineer_HMI.fPGain_IL_Neg;
	fIntegralGain := G_Engineer_HMI.fIGain_IL_Neg;
	fDerivateGain := G_Engineer_HMI.fDGain_IL_Neg;
ELSE
	fProportionalGain := G_Engineer_HMI.fPGain_IL_Pos;
	fIntegralGain := G_Engineer_HMI.fIGain_IL_Pos;
	fDerivateGain := G_Engineer_HMI.fDGain_IL_Pos;
END_IF

		
		fbPID_IL(
	ssMethodType := BOOL_TO_SINT(bEnable),
	fSignalReference := fDisplacementNormalizedInput,
	fSignalFeedback := fYokeNormalizedFeedback,
	fProportionalGain := fProportionalGain,
	fIntegralGain := fIntegralGain,
	bActivateIntegralControl := G_Engineer_HMI.bIenable_IL,
	bEnable := bEnable,
	bIntegralControlReset := NOT(bEnable),
	bActivateDerivativeControl := G_Engineer_HMI.bDenable_IL,
	fDerivativeGain := fDerivateGain,
	fClosedLoopSignal => fNormalizedOutput,
	fSignalError =>G_PID_Tuning.fYoke_error,
	P_out => G_PID_Tuning.fPout_IL,
	I_out => G_PID_Tuning.fIout_IL,
	D_out => G_PID_Tuning.fDout_IL
	);	


	//Make Output global for plot
	G_PID_Tuning.PID_output_IL := fNormalizedOutput;
	
ELSE 
	fNormalizedOutput := 0.0; // Ingen output uten aktivering
END_IF

END_FUNCTION_BLOCK

// ---- Function Blocks/FBs for Motion Control/Ekstra FBs/FB_Target_displacement.TcPOU
FUNCTION_BLOCK FB_Target_displacement
VAR_INPUT
END_VAR
VAR_OUTPUT
	fTarget_dis				: LREAL;
END_VAR
VAR
END_VAR

IF G_Engineer_HMI.bJoystick_slider_active THEN
	G_Engineer_HMI.fDisplacement_target := G_Sensors.fJoystickNormalizedX;
ELSE
G_Engineer_HMI.fDisplacement_target	 := G_Engineer_HMI.fDisplacement_target;		
END_IF

fTarget_dis := G_Engineer_HMI.fDisplacement_target;

END_FUNCTION_BLOCK

// ---- Function Blocks/FBs for Motion Control/Ekstra FBs/FB_ControlReset_SC.TcPOU
FUNCTION_BLOCK FB_ControlReset_SC
VAR_INPUT
	fVelRef			: LREAL;
	ferror			: LREAL;

END_VAR
VAR_OUTPUT
	bReset			: BOOL;
END_VAR
VAR
	ferror_Tolerence	: LREAL := 0.001;
END_VAR

IF fVelRef = 0.0 AND ABS(ferror) < ferror_Tolerence THEN
	bReset := TRUE;
ELSE
	bReset := FALSE;
END_IF

END_FUNCTION_BLOCK

// ---- Function Blocks/FBs for Motion Control/Ekstra FBs/FB_Feedforward_SC.TcPOU
FUNCTION_BLOCK FB_Feedforward_SC
VAR_INPUT
	fVelref			: LREAL;
	fKff			: LREAL;
	fVelref_dot		: LREAL;
END_VAR
VAR_OUTPUT
	fAlpha			: LREAL;
END_VAR
VAR
	fM_0				: LREAL;
	fomega_0			: LREAL;
	x					: LREAL;
	fMFr				: LREAL;
	J_eff				: LREAL;
	fD_Max				: LREAL;
	fdelta_p_Pa			: LREAL;
END_VAR

fM_0 := 53.0;
fomega_0 := 0.005;
x := (fVelref/fomega_0);
J_eff := 0.01 + 0.1 + G_Parameters.stParam.fPayloadMass * G_Parameters.stParam.fWinchDrumRadius * G_Parameters.stParam.fWinchDrumRadius;
fD_Max := 180.0/1000000.0; // cm^3/rev -> *10^-6 m^3/rev
fdelta_p_Pa := G_Sensors.fDeltaPMotor * 100000;

// For å skrive tanh med EXP: https://www.youtube.com/watch?v=r76jFsDXkHw

fMFr := fM_0 * (EXP(2.0 * x) - 1.0)/(EXP(2.0 * x)+1.0);

fAlpha := LIMIT(0.0, fKff*((G_Parameters.stParam.fPayloadMass * 9.81 * G_Parameters.stParam.fWinchDrumRadius + fMFr + J_eff * fVelref_dot)*2.0 * PI)/(fD_Max * LIMIT(10.0,fdelta_p_Pa,200.0)), 1.0);

END_FUNCTION_BLOCK

// ---- Function Blocks/FBs Auto Control/FB_Derivator.TcPOU
FUNCTION_BLOCK FB_Derivator
VAR_INPUT
	Input: LREAL;
	ssMethodType: SINT;
END_VAR
VAR_OUTPUT
	Derivated_output: LREAL;
END_VAR
VAR
	rtb_TSamp: LREAL;
	UD_DSTATE: LREAL;
END_VAR



CASE ssMethodType OF
    0: 
        (* SystemInitialize for Atomic SubSystem: '<Root>/FB_Derivator' *)
        (* InitializeConditions for UnitDelay: '<S2>/UD'
         *
         * Block description for '<S2>/UD':
         *  
         *  Store in Global RAM *)
        UD_DSTATE := 0.0;
        (* End of SystemInitialize for SubSystem: '<Root>/FB_Derivator' *)
    1: 
        (* Outputs for Atomic SubSystem: '<Root>/FB_Derivator' *)
        (* SampleTimeMath: '<S2>/TSamp'
         *
         * About '<S2>/TSamp':
         *  y = u * K where K = 1 / ( w * Ts )
         *   *)
        rtb_TSamp := Input * 100.0;
        (* Outport: '<Root>/Derivated_output' incorporates:
         *  Sum: '<S2>/Diff'
         *  UnitDelay: '<S2>/UD'
         *
         * Block description for '<S2>/Diff':
         *  
         *  Add in CPU
         *
         * Block description for '<S2>/UD':
         *  
         *  Store in Global RAM *)
        Derivated_output := LIMIT(-1.0,rtb_TSamp - UD_DSTATE,1.0);
        (* Update for UnitDelay: '<S2>/UD'
         *
         * Block description for '<S2>/UD':
         *  
         *  Store in Global RAM *)
        UD_DSTATE := rtb_TSamp;
        (* End of Outputs for SubSystem: '<Root>/FB_Derivator' *)
END_CASE;

END_FUNCTION_BLOCK

// ---- Function Blocks/FBs for Motion Control/FB_Auto_SC.TcPOU
FUNCTION_BLOCK FB_Auto_SC
VAR_INPUT
	bEnable				: BOOL;
END_VAR
VAR_OUTPUT
	fPCV				: LREAL;
	fSCV				: LREAL;
	
END_VAR
VAR
	
//Function Blocks
fbPID_OL_startpos				: FB_PID_Controller;
fbPID_OL_sine				: FB_PID_Controller;

fbDeadband_startpos			: FB_Deadband_Auto;
fbDeadband_sine				: FB_Deadband_Auto_sine;

fbDisplacementControl_IL_startpos	: FB_DisplacementControl_SC;
fbDisplacementControl_IL_sine	: FB_DisplacementControl_SC;

fbDerivator					: FB_Derivator;

fbClock						: FB_Clock;
fbSineActivation			: FB_SineActivation_SC;
fbMUX_selector				: FB_MUX_selector;

fbGain_Chooser_P			: FB_GainChooser;
fbGain_Chooser_I			: FB_GainChooser;
fb_ControlReset_startpos	: FB_ControlReset_SC;
fb_ControlReset_sine		:FB_ControlReset_SC;

//Deadband
fDeadbandComp_out			: LREAL;
fDeadbandComp_out_startpos			: LREAL;

//Outer Loop output
fSC_ClosedLoopSingal		: LREAL;
fOuterLoopError				: LREAL;

//Sine Ref signal
fSineRefSignal_SC			: LREAL;
fWinchVelRefSine			: LREAL;

//Valvesignals
fPCV_set					: LREAL := 1.0;
fPCV_On						: LREAL;
fPCV_Off					: LREAL;

fSCV_startpos				: LREAL;
fSCV_sine					: LREAL;
fSCV_Off					: LREAL;


END_VAR
VAR // added by the converter: edge detectors and wires of the graphical bodies
    _w1 : LREAL;
    _w2 : BOOL;
END_VAR

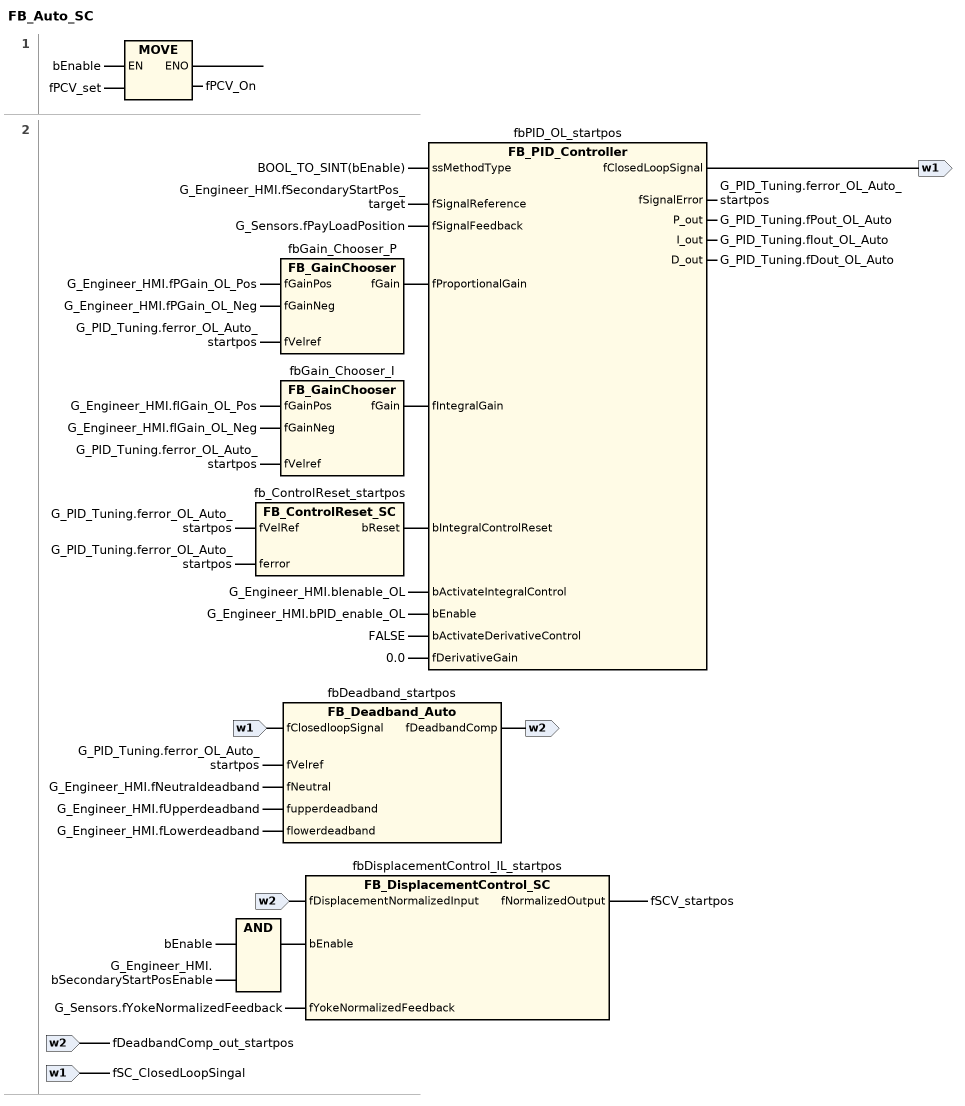
// NETWORK 1
IF bEnable THEN fPCV_On := fPCV_set; END_IF

// NETWORK 2
fbGain_Chooser_P(
    fGainPos := G_Engineer_HMI.fPGain_OL_Pos,
    fGainNeg := G_Engineer_HMI.fPGain_OL_Neg,
    fVelref := G_PID_Tuning.ferror_OL_Auto_startpos); // FB_GainChooser
fbGain_Chooser_I(
    fGainPos := G_Engineer_HMI.fIGain_OL_Pos,
    fGainNeg := G_Engineer_HMI.fIGain_OL_Neg,
    fVelref := G_PID_Tuning.ferror_OL_Auto_startpos); // FB_GainChooser
fb_ControlReset_startpos(fVelRef := G_PID_Tuning.ferror_OL_Auto_startpos, ferror := G_PID_Tuning.ferror_OL_Auto_startpos); // FB_ControlReset_SC
fbPID_OL_startpos(
    ssMethodType := BOOL_TO_SINT(bEnable),
    fSignalReference := G_Engineer_HMI.fSecondaryStartPos_target,
    fSignalFeedback := G_Sensors.fPayLoadPosition,
    fProportionalGain := fbGain_Chooser_P.fGain,
    fIntegralGain := fbGain_Chooser_I.fGain,
    bIntegralControlReset := fb_ControlReset_startpos.bReset,
    bActivateIntegralControl := G_Engineer_HMI.bIenable_OL,
    bEnable := G_Engineer_HMI.bPID_enable_OL,
    bActivateDerivativeControl := FALSE,
    fDerivativeGain := 0.0,
    fSignalError => G_PID_Tuning.ferror_OL_Auto_startpos,
    P_out => G_PID_Tuning.fPout_OL_Auto,
    I_out => G_PID_Tuning.fIout_OL_Auto,
    D_out => G_PID_Tuning.fDout_OL_Auto); // FB_PID_Controller
fbDeadband_startpos(
    fClosedloopSignal := fbPID_OL_startpos.fClosedLoopSignal,
    fVelref := G_PID_Tuning.ferror_OL_Auto_startpos,
    fNeutral := G_Engineer_HMI.fNeutraldeadband,
    fupperdeadband := G_Engineer_HMI.fUpperdeadband,
    flowerdeadband := G_Engineer_HMI.fLowerdeadband); // FB_Deadband_Auto
fbDisplacementControl_IL_startpos(
    fDisplacementNormalizedInput := fbDeadband_startpos.fDeadbandComp,
    bEnable := bEnable AND G_Engineer_HMI.bSecondaryStartPosEnable,
    fYokeNormalizedFeedback := G_Sensors.fYokeNormalizedFeedback); // FB_DisplacementControl_SC
fSCV_startpos := fbDisplacementControl_IL_startpos.fNormalizedOutput;
fDeadbandComp_out_startpos := fbDeadband_startpos.fDeadbandComp;
fSC_ClosedLoopSingal := fbPID_OL_startpos.fClosedLoopSignal;

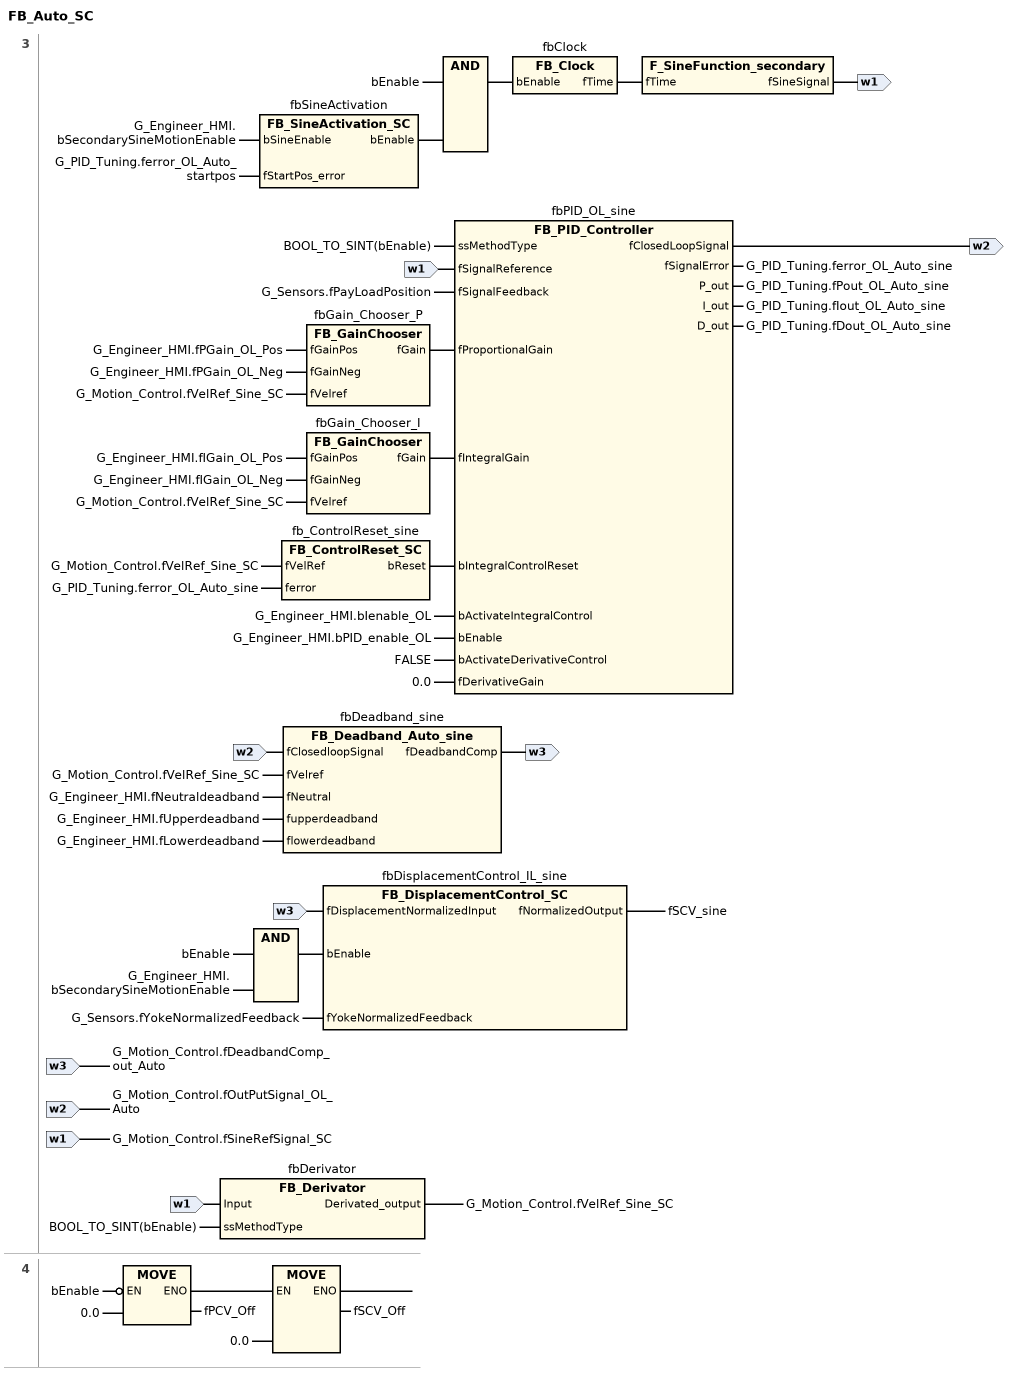
// NETWORK 3
fbSineActivation(bSineEnable := G_Engineer_HMI.bSecondarySineMotionEnable, fStartPos_error := G_PID_Tuning.ferror_OL_Auto_startpos); // FB_SineActivation_SC
fbClock(bEnable := bEnable AND fbSineActivation.bEnable); // FB_Clock
F_SineFunction_secondary(fTime := fbClock.fTime, fSineSignal => _w1);
fbGain_Chooser_P(
    fGainPos := G_Engineer_HMI.fPGain_OL_Pos,
    fGainNeg := G_Engineer_HMI.fPGain_OL_Neg,
    fVelref := G_Motion_Control.fVelRef_Sine_SC); // FB_GainChooser
fbGain_Chooser_I(
    fGainPos := G_Engineer_HMI.fIGain_OL_Pos,
    fGainNeg := G_Engineer_HMI.fIGain_OL_Neg,
    fVelref := G_Motion_Control.fVelRef_Sine_SC); // FB_GainChooser
fb_ControlReset_sine(fVelRef := G_Motion_Control.fVelRef_Sine_SC, ferror := G_PID_Tuning.ferror_OL_Auto_sine); // FB_ControlReset_SC
fbPID_OL_sine(
    ssMethodType := BOOL_TO_SINT(bEnable),
    fSignalReference := _w1,
    fSignalFeedback := G_Sensors.fPayLoadPosition,
    fProportionalGain := fbGain_Chooser_P.fGain,
    fIntegralGain := fbGain_Chooser_I.fGain,
    bIntegralControlReset := fb_ControlReset_sine.bReset,
    bActivateIntegralControl := G_Engineer_HMI.bIenable_OL,
    bEnable := G_Engineer_HMI.bPID_enable_OL,
    bActivateDerivativeControl := FALSE,
    fDerivativeGain := 0.0,
    fSignalError => G_PID_Tuning.ferror_OL_Auto_sine,
    P_out => G_PID_Tuning.fPout_OL_Auto_sine,
    I_out => G_PID_Tuning.fIout_OL_Auto_sine,
    D_out => G_PID_Tuning.fDout_OL_Auto_sine); // FB_PID_Controller
fbDeadband_sine(
    fClosedloopSignal := fbPID_OL_sine.fClosedLoopSignal,
    fVelref := G_Motion_Control.fVelRef_Sine_SC,
    fNeutral := G_Engineer_HMI.fNeutraldeadband,
    fupperdeadband := G_Engineer_HMI.fUpperdeadband,
    flowerdeadband := G_Engineer_HMI.fLowerdeadband); // FB_Deadband_Auto_sine
fbDisplacementControl_IL_sine(
    fDisplacementNormalizedInput := fbDeadband_sine.fDeadbandComp,
    bEnable := bEnable AND G_Engineer_HMI.bSecondarySineMotionEnable,
    fYokeNormalizedFeedback := G_Sensors.fYokeNormalizedFeedback); // FB_DisplacementControl_SC
fSCV_sine := fbDisplacementControl_IL_sine.fNormalizedOutput;
G_Motion_Control.fDeadbandComp_out_Auto := fbDeadband_sine.fDeadbandComp;
G_Motion_Control.fOutPutSignal_OL_Auto := fbPID_OL_sine.fClosedLoopSignal;
G_Motion_Control.fSineRefSignal_SC := _w1;
fbDerivator(Input := _w1, ssMethodType := BOOL_TO_SINT(bEnable)); // FB_Derivator
G_Motion_Control.fVelRef_Sine_SC := fbDerivator.Derivated_output;

// NETWORK 4
_w2 := NOT bEnable;
IF _w2 THEN fPCV_Off := 0.0; END_IF
IF _w2 THEN fSCV_Off := 0.0; END_IF

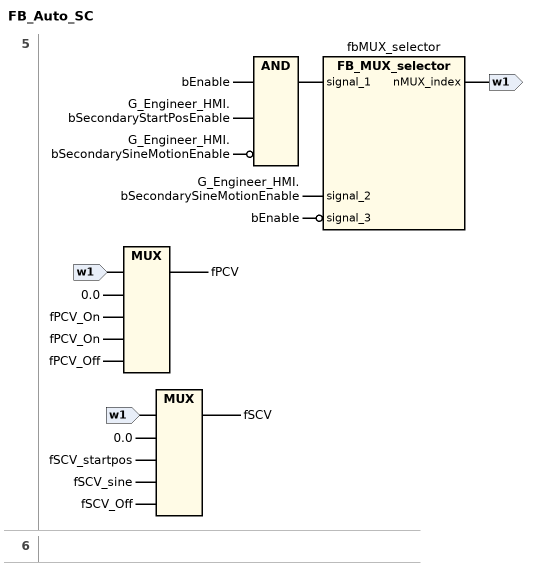
// NETWORK 5
fbMUX_selector(
    signal_1 := bEnable AND G_Engineer_HMI.bSecondaryStartPosEnable AND NOT G_Engineer_HMI.bSecondarySineMotionEnable,
    signal_2 := G_Engineer_HMI.bSecondarySineMotionEnable,
    signal_3 := NOT bEnable); // FB_MUX_selector
fPCV := MUX(fbMUX_selector.nMUX_index, 0.0, fPCV_On, fPCV_On, fPCV_Off);
fSCV := MUX(fbMUX_selector.nMUX_index, 0.0, fSCV_startpos, fSCV_sine, fSCV_Off);

// NETWORK 6

END_FUNCTION_BLOCK

// ---- Function Blocks/Deadband Comp/FB_Deadband_Auto.TcPOU
FUNCTION_BLOCK FB_Deadband_Auto
VAR_INPUT
	fClosedloopSignal	: LREAL;
	fVelref				: LREAL;
	fNeutral			: LREAL;
	fupperdeadband		: LREAL;
	flowerdeadband		: LREAL;
	
END_VAR
VAR_OUTPUT
	fDeadbandComp		: LREAL;
END_VAR
VAR
END_VAR

IF fVelref > 0.01 THEN
	fDeadbandComp := LIMIT(fNeutral,fupperdeadband + fClosedloopSignal,1.0);
ELSIF fVelref < -0.01 THEN
	fDeadbandComp := LIMIT(0.1,flowerdeadband + fClosedloopSignal,fNeutral); //Kanskje minus her men tror input blir - så da blir det fikset
ELSE
	fDeadbandComp := LIMIT(-1.0,fNeutral,1.0);
END_IF

END_FUNCTION_BLOCK

// ---- Function Blocks/Deadband Comp/FB_Deadband_Auto_sine.TcPOU
FUNCTION_BLOCK FB_Deadband_Auto_sine
VAR_INPUT
	fClosedloopSignal	: LREAL;
	fVelref				: LREAL;
	fNeutral			: LREAL;
	fupperdeadband		: LREAL;
	flowerdeadband		: LREAL;
	
END_VAR
VAR_OUTPUT
	fDeadbandComp		: LREAL;
END_VAR
VAR
END_VAR

IF fVelref > 0.0 THEN
	fDeadbandComp := LIMIT(fNeutral,fupperdeadband + fClosedloopSignal,1.0);
ELSIF fVelref < 0.0 THEN
	fDeadbandComp := LIMIT(0.1,flowerdeadband + fClosedloopSignal,fNeutral); //Kanskje minus her men tror input blir - så da blir det fikset
ELSE
	fDeadbandComp := LIMIT(0.1,fNeutral,1.0);
END_IF

END_FUNCTION_BLOCK

// ---- Function Blocks/FBs Auto Control/FB_SineActivation_SC.TcPOU
FUNCTION_BLOCK FB_SineActivation_SC
VAR_INPUT
	bSineEnable			: BOOL;
	fStartPos_error		: LREAL;
END_VAR
VAR_OUTPUT
	bEnable				: BOOL;
END_VAR
VAR
	bStartPosOK			: BOOL;
END_VAR

IF ABS(fStartPos_error) < 0.2 THEN
	bStartPosOK := TRUE;
ELSIF NOT (G_IO.bStartButton) THEN
	bStartPosOK := FALSE;
END_IF

IF NOT(G_IO.bStartButton) THEN
	bEnable := FALSE;
	G_Engineer_HMI.bSecondarySineMotionEnable := FALSE;
	ELSIF bStartPosOK AND bSineEnable THEN
		bEnable := TRUE;
END_IF

END_FUNCTION_BLOCK

// ---- Functions/F_SineFunction_secondary.TcPOU
FUNCTION F_SineFunction_secondary : LREAL
VAR_INPUT
	fTime 				: LREAL;
END_VAR
VAR_OUTPUT
	fSineSignal 		: LREAL;
END_VAR
VAR
	u					: LREAL;
	ft_ENV				: LREAL := 3.0;
	y					: LREAL;
	
END_VAR

(*u := fTime/ft_ENV;

IF u > 1.0 THEN
	u := 1.0;
END_IF

y := (3.0*u*u) - (2.0*u*u*u);*)

fSineSignal := G_Engineer_HMI.fAmp * SIN(2.0 * PI * G_Engineer_HMI.fFreq * fTime) + G_Engineer_HMI.fSinemidpoint; //y gange i starten om soft start skal på

END_FUNCTION

// ---- Function Blocks/FBs for Motion Control/FB_Auto_Combination.TcPOU
FUNCTION_BLOCK FB_Auto_Combination
VAR_INPUT
	bEnable					: BOOL;
END_VAR
VAR_OUTPUT
	fPCV					: LREAL;
	fSCV					: LREAL;
END_VAR
VAR

//Sine Wave
fbClock						: FB_Clock;	
fSineRef					: LREAL;

//Off
fPCV_Off					: LREAL;
fSCV_Off					: LREAL;


//////Primary Control////////
fSCV_On						: LREAL;
fPCV_PC						: LREAL;
	
fbAutoSineMotion_PC			: FB_AutoSineMotion;

/////Secondary Control/////
fPCV_set					: LREAL := 1.0;
fPCV_On						: LREAL;
fSCV_SC						: LREAL;

fbGain_Chooser_P			: FB_GainChooser;
fbGain_Chooser_I			: FB_GainChooser;
fbDerivator					: FB_Derivator;

fbPID_OL					: FB_PID_Controller;
fbDeadband_sine				: FB_Deadband_Auto_sine;
fbDisplacementControl_IL	: FB_DisplacementControl_SC;



//Plotting
fVelref_sine				: LREAL;
fOutPutSignal_OL_combi		: LREAL;
fDeadbandComp_out			: LREAL;

//MUX
fbMUX_selector				: FB_MUX_selector;

END_VAR
VAR // added by the converter: edge detectors and wires of the graphical bodies
    _w1 : LREAL;
    _w2 : BOOL;
END_VAR

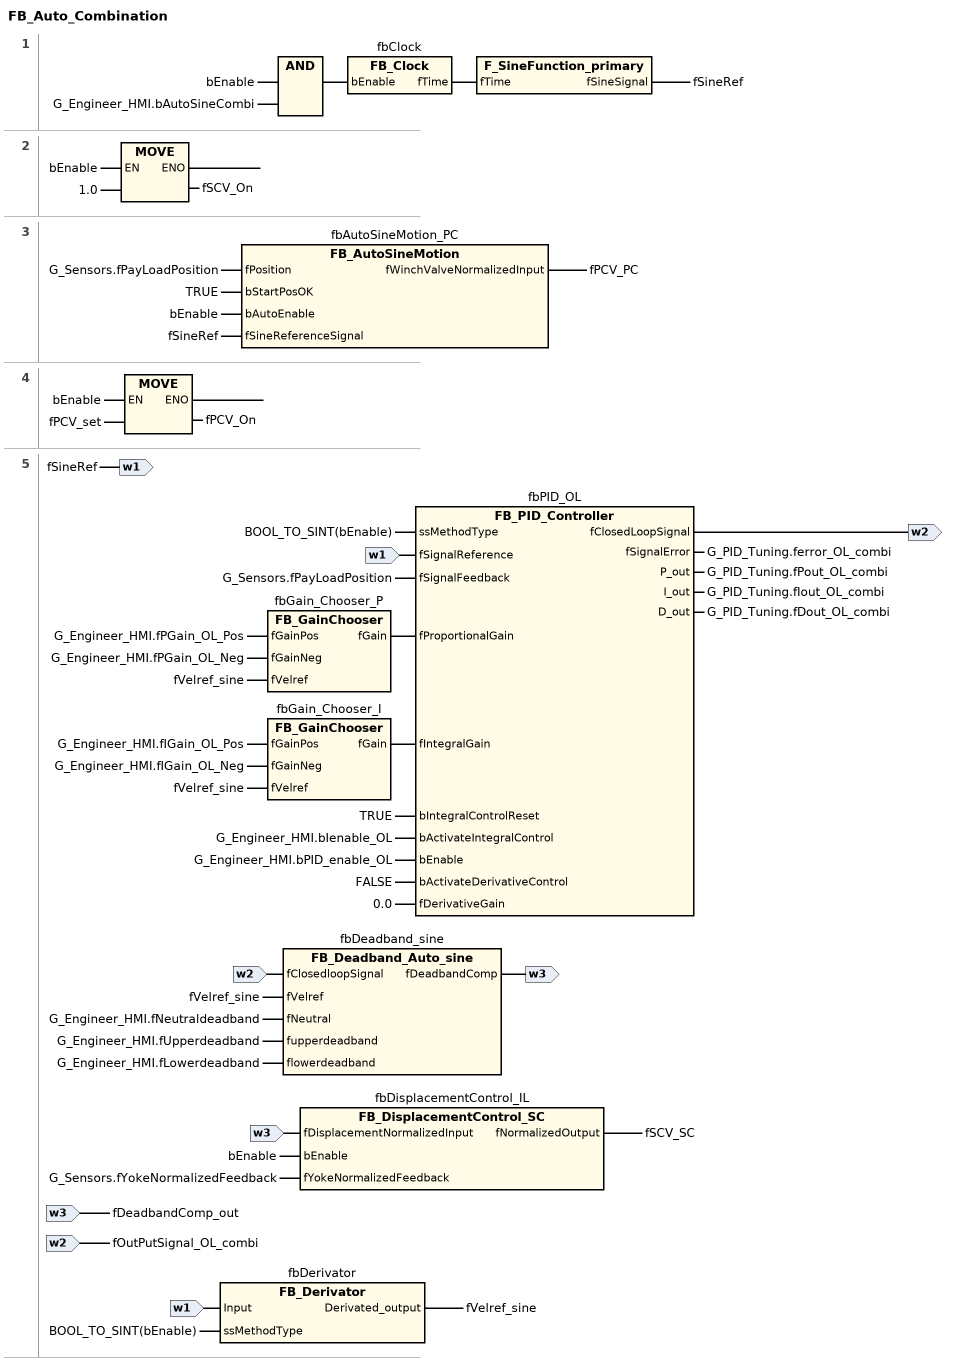
// NETWORK 1
fbClock(bEnable := bEnable AND G_Engineer_HMI.bAutoSineCombi); // FB_Clock
F_SineFunction_primary(fTime := fbClock.fTime, fSineSignal => _w1);
fSineRef := _w1;

// NETWORK 2
IF bEnable THEN fSCV_On := 1.0; END_IF

// NETWORK 3
fbAutoSineMotion_PC(
    fPosition := G_Sensors.fPayLoadPosition,
    bStartPosOK := TRUE,
    bAutoEnable := bEnable,
    fSineReferenceSignal := fSineRef); // FB_AutoSineMotion
fPCV_PC := fbAutoSineMotion_PC.fWinchValveNormalizedInput;

// NETWORK 4
IF bEnable THEN fPCV_On := fPCV_set; END_IF

// NETWORK 5
fbGain_Chooser_P(
    fGainPos := G_Engineer_HMI.fPGain_OL_Pos,
    fGainNeg := G_Engineer_HMI.fPGain_OL_Neg,
    fVelref := fVelref_sine); // FB_GainChooser
fbGain_Chooser_I(
    fGainPos := G_Engineer_HMI.fIGain_OL_Pos,
    fGainNeg := G_Engineer_HMI.fIGain_OL_Neg,
    fVelref := fVelref_sine); // FB_GainChooser
fbPID_OL(
    ssMethodType := BOOL_TO_SINT(bEnable),
    fSignalReference := fSineRef,
    fSignalFeedback := G_Sensors.fPayLoadPosition,
    fProportionalGain := fbGain_Chooser_P.fGain,
    fIntegralGain := fbGain_Chooser_I.fGain,
    bIntegralControlReset := TRUE,
    bActivateIntegralControl := G_Engineer_HMI.bIenable_OL,
    bEnable := G_Engineer_HMI.bPID_enable_OL,
    bActivateDerivativeControl := FALSE,
    fDerivativeGain := 0.0,
    fSignalError => G_PID_Tuning.ferror_OL_combi,
    P_out => G_PID_Tuning.fPout_OL_combi,
    I_out => G_PID_Tuning.fIout_OL_combi,
    D_out => G_PID_Tuning.fDout_OL_combi); // FB_PID_Controller
fbDeadband_sine(
    fClosedloopSignal := fbPID_OL.fClosedLoopSignal,
    fVelref := fVelref_sine,
    fNeutral := G_Engineer_HMI.fNeutraldeadband,
    fupperdeadband := G_Engineer_HMI.fUpperdeadband,
    flowerdeadband := G_Engineer_HMI.fLowerdeadband); // FB_Deadband_Auto_sine
fbDisplacementControl_IL(
    fDisplacementNormalizedInput := fbDeadband_sine.fDeadbandComp,
    bEnable := bEnable,
    fYokeNormalizedFeedback := G_Sensors.fYokeNormalizedFeedback); // FB_DisplacementControl_SC
fSCV_SC := fbDisplacementControl_IL.fNormalizedOutput;
fDeadbandComp_out := fbDeadband_sine.fDeadbandComp;
fOutPutSignal_OL_combi := fbPID_OL.fClosedLoopSignal;
fbDerivator(Input := fSineRef, ssMethodType := BOOL_TO_SINT(bEnable)); // FB_Derivator
fVelref_sine := fbDerivator.Derivated_output;

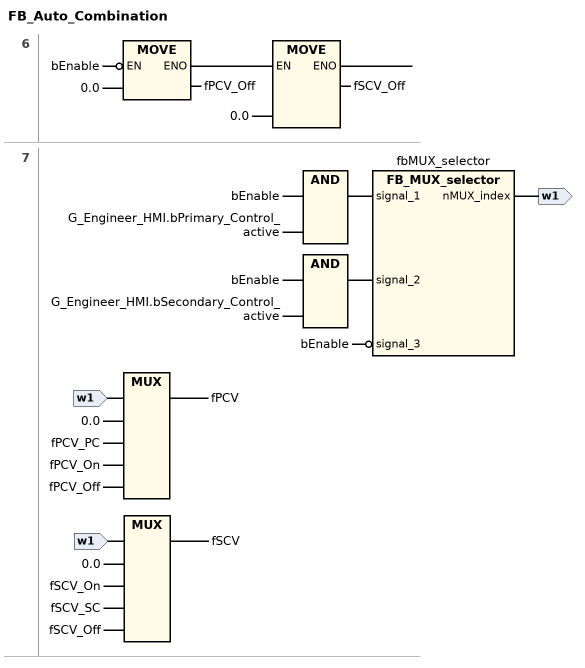
// NETWORK 6
_w2 := NOT bEnable;
IF _w2 THEN fPCV_Off := 0.0; END_IF
IF _w2 THEN fSCV_Off := 0.0; END_IF

// NETWORK 7
fbMUX_selector(
    signal_1 := bEnable AND G_Engineer_HMI.bPrimary_Control_active,
    signal_2 := bEnable AND G_Engineer_HMI.bSecondary_Control_active,
    signal_3 := NOT bEnable); // FB_MUX_selector
fPCV := MUX(fbMUX_selector.nMUX_index, 0.0, fPCV_PC, fPCV_On, fPCV_Off);
fSCV := MUX(fbMUX_selector.nMUX_index, 0.0, fSCV_On, fSCV_SC, fSCV_Off);

END_FUNCTION_BLOCK

// ---- Function Blocks/FBs for Motion Control/FB_EndStop.TcPOU
FUNCTION_BLOCK FB_EndStop
VAR_INPUT
	//Trenger denne enable???
	//Skal de settes til 0 her når de ikke brukes?? må det gjøres en plass??
	fPCV				: LREAL;
	fSCV				: LREAL;
END_VAR
VAR_OUTPUT
	fPCV_norm_input		: LREAL;
	fSCV_norm_input		: LREAL;
END_VAR
VAR
u_Neg					: LREAL;
y_Neg					: LREAL;
u_Pos					: LREAL;
y_Pos					: LREAL;

END_VAR

//////////Soft Stop////////////
u_Neg := LIMIT(0,((G_Sensors.fPayLoadPosition - G_Parameters.stParam.fWinchEndStopNeg ) / ( G_Parameters.stParam.fWinchEndStopNeg_soft -  G_Parameters.stParam.fWinchEndStopNeg)),1);

y_Neg :=  LIMIT(0.1,((3.0*u_Neg*u_Neg)-(2.0*u_Pos*u_Pos*u_Pos)),1);

u_Pos := LIMIT(0,((G_Sensors.fPayLoadPosition - G_Parameters.stParam.fWinchEndStopPos ) / ( G_Parameters.stParam.fWinchEndStopPos_soft -  G_Parameters.stParam.fWinchEndStopPos)),1);

y_Pos :=  LIMIT(0.1,((3.0*u_Pos*u_Pos)-(2.0*u_Pos*u_Pos*u_Pos)),1);

//////////End Stop///////////// skal lage FB på dette
IF G_Sensors.fPayLoadPosition < G_Parameters.stParam.fWinchEndStopNeg_soft AND  G_Sensors.fPayLoadPosition > G_Parameters.stParam.fWinchEndStopNeg AND NOT (G_Engineer_HMI.bEndStopOverride) THEN
	fPCV_norm_input := LIMIT(-1.0, y_Neg*fPCV, 1.0);

ELSIF G_Sensors.fPayLoadPosition < G_Parameters.stParam.fWinchEndStopNeg AND NOT (G_Engineer_HMI.bEndStopOverride) THEN
	G_Engineer_HMI.bEndStopUpActive := FALSE;
	G_Engineer_HMI.bEndStopDownActive := TRUE;
	fPCV_norm_input := LIMIT(0.0, fPCV, 1.0);
	
ELSIF 	G_Sensors.fPayLoadPosition > G_Parameters.stParam.fWinchEndStopPos_soft AND  G_Sensors.fPayLoadPosition < G_Parameters.stParam.fWinchEndStopPos AND NOT (G_Engineer_HMI.bEndStopOverride) THEN
	fPCV_norm_input := LIMIT(-1.0, y_Pos*fPCV, 1.0);
	
ELSIF G_Sensors.fPayLoadPosition > G_Parameters.stParam.fWinchEndStopPos AND NOT (G_Engineer_HMI.bEndStopOverride) THEN
	G_Engineer_HMI.bEndStopUpActive := TRUE;
	G_Engineer_HMI.bEndStopDownActive := FALSE;
	fPCV_norm_input := LIMIT(-1.0, fPCV, 0.0);
ELSE
	G_Engineer_HMI.bEndStopUpActive := FALSE;
	G_Engineer_HMI.bEndStopDownActive := FALSE;
	fPCV_norm_input := LIMIT(-1.0, fPCV, 1.0);
END_IF


fSCV_norm_input := LIMIT(-1, fSCV, 1);

//Ikke lagt inn men forslag til endstop logikk:
//Sette SCV til en når den når endestoppne (når SCV er 1 og PCV er 0 kan den trygt styres ut av området

END_FUNCTION_BLOCK

// ---- Function Blocks/FBs for Motion Control/FB_Outputs.TcPOU

FUNCTION_BLOCK FB_Outputs
VAR_INPUT
	fWinchValveNormalizedInput		: LREAL;
	fDisplacementControlSignal		: LREAL; //Dette er signalet som endrer displacement
END_VAR
VAR_OUTPUT
	fPCV_raw							: INT;
	fSCV_raw							: INT;
END_VAR
VAR
	bEnableMotion					: BOOL;

//Winch
bEnableWinch   					: BOOL;  
bEnableValveOutputWinch			: BOOL;

//Displacement
fDisplacementNormalizedInput	: LREAL ; //Kan fra Controlsignal til denne på displacement slik det blir likt som på winch
										  // lar det stå for å unngå forvirring i starteb

bEnableValveOutputDisp	 		: BOOL;

//Function Blocks
fbWinchValveOutput				: FB_ValveOutput;
fbDisplacementValveOutput		: FB_DisplacementValveOutput;
	
	
END_VAR

IF MAIN.eStatus = E_Status.Running THEN
	G_IO.bEnablePCDV := TRUE;
	G_IO.bWinchValveEnable := TRUE;
ELSE
	G_IO.bEnablePCDV := FALSE;	
	G_IO.bWinchValveEnable := FALSE;
END_IF

////////////////Enable Motion logic/////////////////////////
IF ((P_MotionControl.bAutoEnable_SC OR P_MotionControl.bAutoEnable_PC) AND G_IO.bStartButton) OR ((P_MotionControl.bManualEnable_PC OR P_MotionControl.bManualEnable_SC) AND G_IO.bWinchEnable) THEN
	bEnableMotion := TRUE;
ELSE 
	bEnableMotion := FALSE; 
END_IF

//////////////Winch////////////////
IF (MAIN.eStatus = E_Status.Running) AND bEnableMotion THEN
	G_IO.bOpenBrakes := TRUE; 
	bEnableWinch := TRUE; 
 ELSE 
	 G_IO.bOpenBrakes := FALSE; 
	 bEnableWinch := FALSE; 
END_IF



//////PCV output//////
fbWinchValveOutput(
	bEnable := bEnableWinch,
	bDeadBandCompOn := G_Parameters.stParam.bWinchDeadBandCompOn,
	stValveDeadBand := G_Parameters.stParam.stWinchValveDeadBand,
	fNormalizedInput := fWinchValveNormalizedInput,
	bEnableValveOutput => bEnableValveOutputWinch,
	nOutput => G_IO.fWinchValveOut
);
fPCV_raw := G_IO.fWinchValveOut;

//////////////Displacement/////////

/////////SCV output///////////

fbDisplacementValveOutput(
	bEnable := (MAIN.eStatus = E_Status.Running),
	bDeadBandCompOn := G_Parameters.stParam.bDisplacementDeadBandCompOn,
	stValveDeadBand := G_Parameters.stParam.stDisplacementValveDeadBand,
	fNormalizedInput := fDisplacementControlSignal,
	bEnableValveOutput => bEnableValveOutputDisp,
	nOutput => G_IO.fWinchPDCVOut
);
fSCV_raw := G_IO.fWinchPDCVOut;

//IF Manual or Auto is not selected valveoutput is set to 0.0 kan fjernes om det aldri blir et problem
//Noe slik på kanskje legges i Motion Control
(*IF NOT (P_MotionControl.bAutoEnable_PC OR P_MotionControl.bManualEnable_SC) AND NOT (P_MotionControl.bManualEnable_PC OR P_MotionControl.bManualEnable_SC) THEN
	fWinchValveInput := 0.0;
END_IF*)

//Styring av displacement med pådrag fra joystick er ikke lagt til

END_FUNCTION_BLOCK

// ---- Function Blocks/FB_DisplacementValveOutput.TcPOU
FUNCTION_BLOCK FB_DisplacementValveOutput
VAR_INPUT
	bEnable : BOOL; 
	bDeadbandCompOn : BOOL; 
	stValveDeadBand : ST_ValveDeadBand; 
	fNormalizedInput : LREAL; 
END_VAR
VAR_OUTPUT
	bEnableValveOutput : BOOL; 
	nOutput : INT; 
END_VAR
VAR
	nOffset : INT := 0; 
	nMaxValue : INT := 10000; 
	nMinValue : INT := -10000;
	nTempOutput : INT; 
END_VAR

IF bDeadbandCompOn THEN 
	IF fNormalizedInput > 0.0 THEN
		nTempOutput := LREAL_TO_INT(fNormalizedInput*(stValveDeadBand.fPosMax - stValveDeadBand.fPosMin) + stValveDeadBand.fPosMin);
	ELSIF fNormalizedInput < 0.0 THEN
		nTempOutput := LREAL_TO_INT(fNormalizedInput*(stValveDeadBand.fNegMax - stValveDeadBand.fNegMin) - stValveDeadBand.fNegMin); 
	ELSE
		nTempOutput := 0; 
	END_IF
	
ELSE 
	IF fNormalizedInput > 0.0 THEN 
		nTempOutput := LREAL_TO_INT(fNormalizedInput*10000.0); // Hvorfor dette? 
	ELSIF fNormalizedInput < 0.0 THEN
		nTempOutput := LREAL_TO_INT(fNormalizedInput*(10000.0)); // Denne skal vel være negativ
	ELSE
		nTempOutput := 0; 
	END_IF
END_IF

IF bEnable THEN
	nOutput := LIMIT(nMinValue, nTempOutput, nMaxValue); 
	bEnableValveOutput := TRUE; 
ELSE
	nOutput := 0;
	bEnableValveOutput := FALSE; 
END_IF

END_FUNCTION_BLOCK

// ---- POUs/P_Outputs.TcPOU
PROGRAM P_Outputs
VAR 
bEnableMotion					: BOOL;

//Winch
bEnableWinch   					: BOOL;  
fWinchValveInput 				: LREAL; 
bEnableValveOutputWinch			: BOOL;
fWinchValveNormalizedInput		: LREAL;

//Displacement
bEnableDisplacement 			: BOOL;  
fDisplacementNormalizedInput	: LREAL := 1.0; //Dette er en start verdi for primærstyring slik at Yoke står på 1
fDisplacementControlSignal		: LREAL; //Dette er signalet som endrer displacement
bEnableValveOutputDisp	 		: BOOL;
fDisplacementControl_output		: LREAL;

//Function Blocks
fbWinchValveOutput				: FB_ValveOutput;
fbDisplacementValveOutput		: FB_DisplacementValveOutput;
fbDisplacementControl			: FB_DisplacementControl;


//Soft End stop legge i FB senere
u_Neg								: LREAL;
y_Neg								: LREAL;
u_Pos								: LREAL;
y_Pos								: LREAL;



//StepInput displacement
T1s									: TIME := T#1S;
fbClock								: FB_Clock;
fStepTime							: LREAL;
END_VAR

IF MAIN.eStatus = E_Status.Running THEN
	G_IO.bEnablePCDV := TRUE;
	G_IO.bWinchValveEnable := TRUE;
ELSE
	G_IO.bEnablePCDV := FALSE;	
	G_IO.bWinchValveEnable := FALSE;
END_IF

////////////////Enable Motion logic/////////////////////////
IF P_MotionControl.bAutoEnable OR ((P_MotionControl.bManualEnable OR P_MotionControl.bSecondaryManualEnable) AND G_IO.bWinchEnable) THEN
	bEnableMotion := TRUE;
ELSE 
		bEnableMotion := FALSE; 
END_IF

//////////////Winch////////////////
IF (MAIN.eStatus = E_Status.Running) AND bEnableMotion THEN
	G_IO.bOpenBrakes := TRUE; 
	bEnableWinch := TRUE; 
 ELSE 
	 G_IO.bOpenBrakes := FALSE; 
	 bEnableWinch := FALSE; 
END_IF

///Choose type of Manual control
IF G_Engineer_HMI.bManualControl_enable AND P_MotionControl.bManualEnable THEN
	fWinchValveInput := LIMIT(-1,G_Motion_Control.fWinchValveInput_joystick_posref,1);
ELSIF P_MotionControl.bManualEnable AND G_Engineer_HMI.bPrimary_Control_active THEN //vurdere om denne skal være elsif eller bare else
	fWinchValveInput := G_Sensors.fJoystickNormalizedY;
ELSIF  P_MotionControl.bSecondaryManualEnable AND G_Engineer_HMI.bSecondary_Control_active THEN
	fWinchValveInput := 1.0;
END_IF

////////Primary Auto Sine Motion////////
(*IF P_MotionControl.bAutoEnable  THEN
	IF G_Engineer_HMI.bAutoStartPosEnable THEN
		fWinchValveInput := G_Motion_Control.fWinchValveNormalizedInput;
		IF P_MotionControl.bStartPosOK THEN
			G_Engineer_HMI.bAutoStartPosEnable := FALSE;
			G_Engineer_HMI.bAutoSineMotionEnable := TRUE;
		END_IF
	ELSIF G_Engineer_HMI.bAutoSineMotionEnable THEN
		fWinchValveInput := G_Motion_Control.fWinchValveNormalizedInput_sine;
	END_IF
END_IF*)

IF P_MotionControl.bAutoEnable  AND G_Engineer_HMI.bAutoStartPosEnable THEN
	fWinchValveInput := G_Motion_Control.fWinchValveNormalizedInput;
END_IF

IF P_MotionControl.bAutoEnable  AND G_Engineer_HMI.bAutoSineMotionEnable THEN
	fWinchValveInput := G_Motion_Control.fWinchValveNormalizedInput_sine;
END_IF



//IF Manual or Auto is not selected valveoutput is set to 0.0 kan fjernes om det aldri blir et problem
IF NOT (P_MotionControl.bAutoEnable OR P_MotionControl.bSecondaryAutoEnable) AND NOT (P_MotionControl.bManualEnable OR P_MotionControl.bSecondaryManualEnable) THEN
	fWinchValveInput := 0.0;
END_IF

//////////Soft Stop////////////
u_Neg := LIMIT(0,((G_Sensors.fPayLoadPosition - G_Parameters.stParam.fWinchEndStopNeg ) / ( G_Parameters.stParam.fWinchEndStopNeg_soft -  G_Parameters.stParam.fWinchEndStopNeg)),1);

y_Neg :=  LIMIT(0.1,((3.0*u_Neg*u_Neg)-(2.0*u_Pos*u_Pos*u_Pos)),1);

u_Pos := LIMIT(0,((G_Sensors.fPayLoadPosition - G_Parameters.stParam.fWinchEndStopPos ) / ( G_Parameters.stParam.fWinchEndStopPos_soft -  G_Parameters.stParam.fWinchEndStopPos)),1);

y_Pos :=  LIMIT(0.1,((3.0*u_Pos*u_Pos)-(2.0*u_Pos*u_Pos*u_Pos)),1);

//////////End Stop///////////// skal lage FB på dette
IF G_Sensors.fPayLoadPosition < G_Parameters.stParam.fWinchEndStopNeg_soft AND  G_Sensors.fPayLoadPosition > G_Parameters.stParam.fWinchEndStopNeg AND NOT (G_Engineer_HMI.bEndStopOverride) THEN
	fWinchValveNormalizedInput := LIMIT(-1.0, y_Neg*fWinchValveInput, 1.0);

ELSIF G_Sensors.fPayLoadPosition < G_Parameters.stParam.fWinchEndStopNeg AND NOT (G_Engineer_HMI.bEndStopOverride) THEN
	G_Engineer_HMI.bEndStopUpActive := FALSE;
	G_Engineer_HMI.bEndStopDownActive := TRUE;
	fWinchValveNormalizedInput := LIMIT(0.0, fWinchValveInput, 1.0);
	
ELSIF 	G_Sensors.fPayLoadPosition > G_Parameters.stParam.fWinchEndStopPos_soft AND  G_Sensors.fPayLoadPosition < G_Parameters.stParam.fWinchEndStopPos AND NOT (G_Engineer_HMI.bEndStopOverride) THEN
	fWinchValveNormalizedInput := LIMIT(-1.0, y_Pos*fWinchValveInput, 1.0);
	
ELSIF G_Sensors.fPayLoadPosition > G_Parameters.stParam.fWinchEndStopPos AND NOT (G_Engineer_HMI.bEndStopOverride) THEN
	G_Engineer_HMI.bEndStopUpActive := TRUE;
	G_Engineer_HMI.bEndStopDownActive := FALSE;
	fWinchValveNormalizedInput := LIMIT(-1.0, fWinchValveInput, 0.0);
ELSE
	G_Engineer_HMI.bEndStopUpActive := FALSE;
	G_Engineer_HMI.bEndStopDownActive := FALSE;
	fWinchValveNormalizedInput := fWinchValveInput;
END_IF

fbWinchValveOutput(
	bEnable := bEnableWinch,
	bDeadBandCompOn := G_Parameters.stParam.bWinchDeadBandCompOn,
	stValveDeadBand := G_Parameters.stParam.stWinchValveDeadBand,
	fNormalizedInput := fWinchValveNormalizedInput,
	bEnableValveOutput => bEnableValveOutputWinch,
	nOutput => G_IO.fWinchValveOut
);


//////////////Displacement/////////
IF (MAIN.eStatus = E_Status.Running) AND G_IO.bDisplacementEnable THEN 
	bEnableDisplacement := TRUE;
ELSE
	bEnableDisplacement := FALSE;
END_IF



fbDisplacementControl(
	bEnable := G_Engineer_HMI.bDisplacement_target_active AND MAIN.eStatus = E_Status.Running,
	fDisplacementNormalizedInput := G_Engineer_HMI.fDisplacement_target,
	fYokeNormalizedFeedback := G_Sensors.fYokeNormalizedFeedback,
	fNormalizedOutput => fDisplacementControl_output
	);



//Dette avgjør hvilket pådrag som skal sendes til DCV
IF bEnableDisplacement THEN
	fDisplacementControlSignal := G_Sensors.fJoystickNormalizedY;
ELSIF G_Engineer_HMI.bDisplacement_target_active THEN
	fDisplacementControlSignal := fDisplacementControl_output;
ELSIF G_Engineer_HMI.bManual_Secondary_joyposref_enable THEN
	fDisplacementControlSignal := LIMIT(-1.0,G_Motion_Control.fSCVInput_joystick_posref_secondary,1.0);
ELSIF G_Engineer_HMI.bStepInput THEN
		fbClock(
			bEnable := G_Engineer_HMI.bStartStepInput,
			fTime => fStepTime
			);
		IF fStepTime < G_Engineer_HMI.fDuration AND G_Engineer_HMI.bStartStepInput THEN
			fDisplacementControlSignal := G_Engineer_HMI.fStepInput / 10000.0;
			
		ELSE
			fDisplacementControlSignal := 0.0;
			G_Engineer_HMI.bStartStepInput := FALSE;
		END_IF
ELSE	
	fDisplacementControlSignal := fDisplacementNormalizedInput;
END_IF

/////////Displacement Control///////////

//For å justere med x akse
IF G_Engineer_HMI.bJoystick_slider_active THEN
	G_Engineer_HMI.fDisplacement_target := LIMIT(0.0,G_Sensors.fJoystickNormalizedX,1.0);
	
	
END_IF


fbDisplacementValveOutput(
	bEnable := (MAIN.eStatus = E_Status.Running),
	bDeadBandCompOn := G_Parameters.stParam.bDisplacementDeadBandCompOn,
	stValveDeadBand := G_Parameters.stParam.stDisplacementValveDeadBand,
	fNormalizedInput := fDisplacementControlSignal,
	bEnableValveOutput => bEnableValveOutputDisp,
	nOutput => G_IO.fWinchPDCVOut
);

END_PROGRAM

// ---- Function Blocks/Currently not in use/FB_EncoderScaling.TcPOU
FUNCTION_BLOCK FB_EncoderScaling
VAR_INPUT
	fPosition							: LREAL;
END_VAR
VAR_OUTPUT
	fNormalizedPosition					: LREAL;
END_VAR
VAR
	
	fWinchEndUp_encoder					: LREAL := G_Parameters.stParam.fWinchEndStopPos;
	fWinchEndDown_encoder				: LREAL := G_Parameters.stParam.fWinchEndStopNeg;
END_VAR


fNormalizedPosition := LIMIT(0,( fPosition - fWinchEndDown_encoder) / (fWinchEndUp_encoder - fWinchEndDown_encoder), 1);
G_Sensors.fWinchEncoderPositionNormalized := fNormalizedPosition;

END_FUNCTION_BLOCK

// ---- Function Blocks/Currently not in use/FB_Motion_Control.TcPOU
FUNCTION_BLOCK FB_Motion_Control
VAR_INPUT
	eStatus : E_Status := E_Status.Checking;
END_VAR
VAR_OUTPUT
	bAutoEnable 							: BOOL;
	bManualEnable 							: BOOL; 
	bSecondaryAutoEnable 					: BOOL; 
	bSecondaryManualEnable				    : BOOL; 

END_VAR
VAR
	fbEncoderScaling 						: FB_EncoderScaling;
	fbAutoStartPos							: FB_AutoStartPos;
	fbAutoSineMotion    					: FB_AutoSineMotion; 
	fbClock_MOOG							: FB_Clock;
	fbClock_dis								: FB_Clock;
	fbDisplacementControl  					: FB_DisplacementControl;
	fbSecondaryControlStartPos				: FB_SecondaryControlStartPos;
	fbJoystick 								: FB_Joystick; 
	fbGetStartPos 							: FB_StartPos;
	fbWinchVelIntegrator					: FB_Integrator;  
	bStartPosOK								: BOOL;
	fWinchVelRefManual						: LREAL; 
	fWinchVelRefAuto                        : LREAL; 
	fWinchPosRefManual						: LREAL; 
	fInitialWinchPos						: LREAL; 
	fbPIDController							: FB_PID_controller_old; 
	
	
	//Secondary control
	
	fbPID 									: FB_PID_controller_old;
	fbFeedForward							: FB_FeedForward;
	
	I_output								: LREAL;
	D_output								: LREAL;
END_VAR
VAR // added by the converter: edge detectors and wires of the graphical bodies
    _w1, _w2 : LREAL;
END_VAR

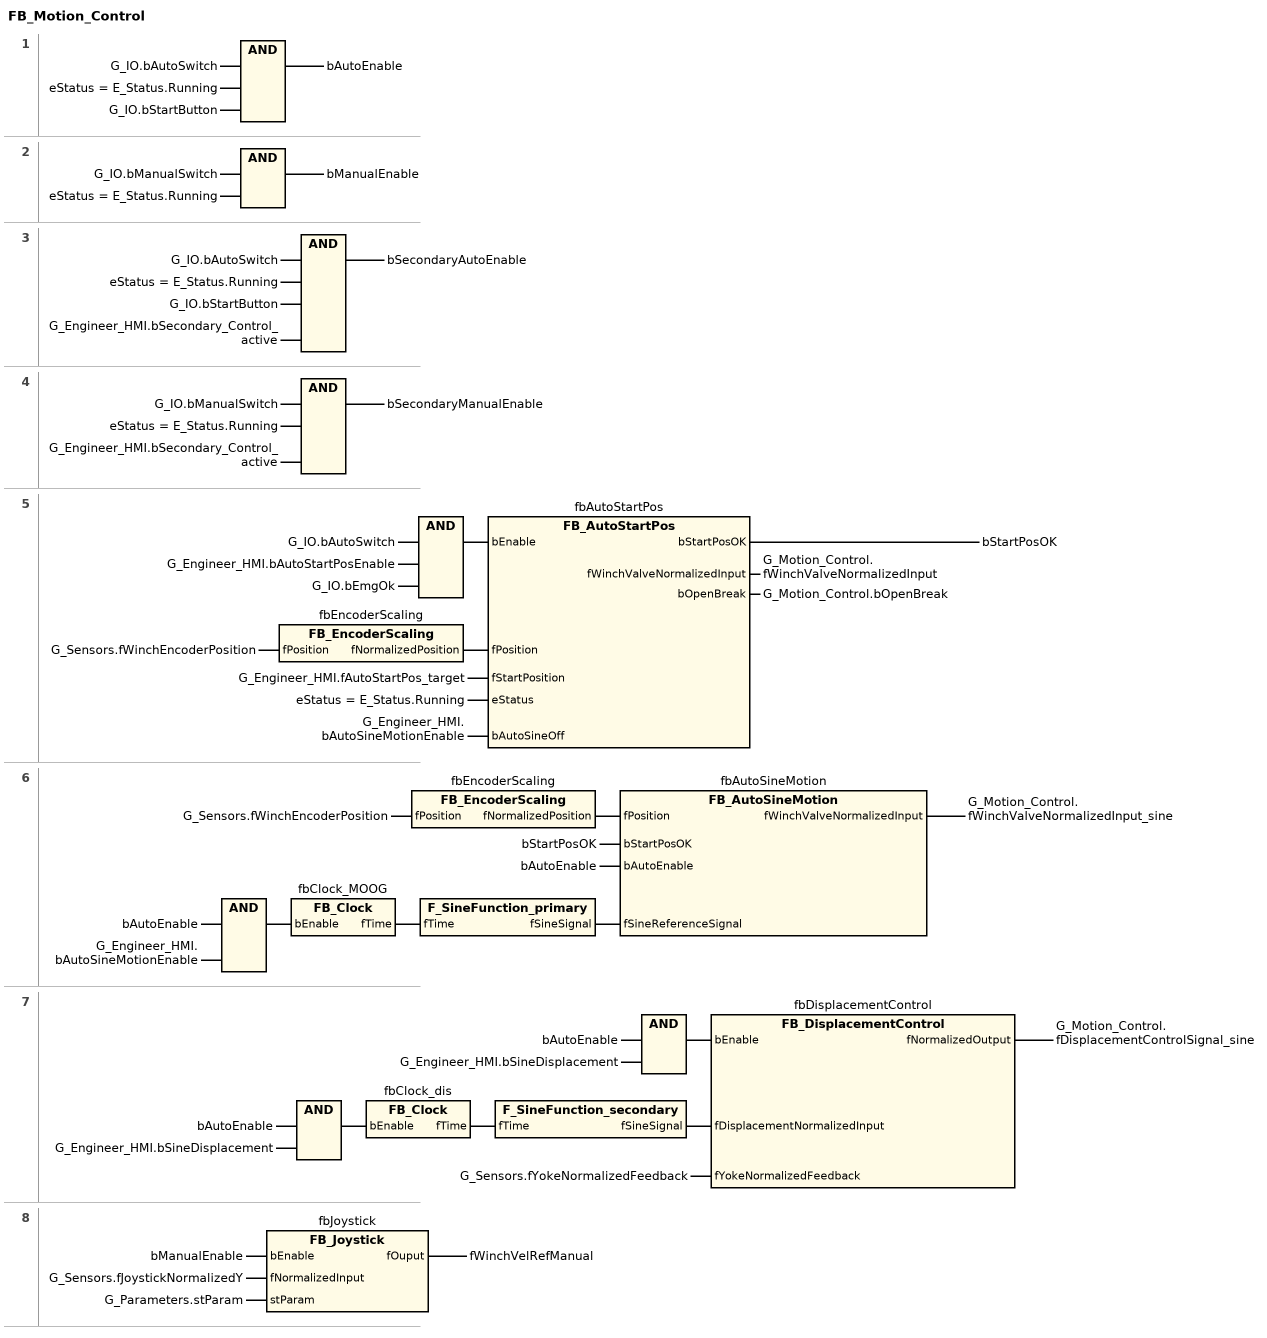
// NETWORK 1
bAutoEnable := G_IO.bAutoSwitch AND (eStatus = E_Status.Running) AND G_IO.bStartButton;

// NETWORK 2
bManualEnable := G_IO.bManualSwitch AND (eStatus = E_Status.Running);

// NETWORK 3
bSecondaryAutoEnable := G_IO.bAutoSwitch AND (eStatus = E_Status.Running) AND G_IO.bStartButton AND G_Engineer_HMI.bSecondary_Control_active;

// NETWORK 4
bSecondaryManualEnable := G_IO.bManualSwitch AND (eStatus = E_Status.Running) AND G_Engineer_HMI.bSecondary_Control_active;

// NETWORK 5
fbEncoderScaling(fPosition := G_Sensors.fWinchEncoderPosition); // FB_EncoderScaling
fbAutoStartPos(
    bEnable := G_IO.bAutoSwitch AND G_Engineer_HMI.bAutoStartPosEnable AND G_IO.bEmgOk,
    fPosition := fbEncoderScaling.fNormalizedPosition,
    fStartPosition := G_Engineer_HMI.fAutoStartPos_target,
    eStatus := eStatus = E_Status.Running,
    bAutoSineOff := G_Engineer_HMI.bAutoSineMotionEnable,
    fWinchValveNormalizedInput => G_Motion_Control.fWinchValveNormalizedInput,
    bOpenBreak => G_Motion_Control.bOpenBreak); // FB_AutoStartPos
bStartPosOK := fbAutoStartPos.bStartPosOK;

// NETWORK 6
fbEncoderScaling(fPosition := G_Sensors.fWinchEncoderPosition); // FB_EncoderScaling
fbClock_MOOG(bEnable := bAutoEnable AND G_Engineer_HMI.bAutoSineMotionEnable); // FB_Clock
F_SineFunction_primary(fTime := fbClock_MOOG.fTime, fSineSignal => _w1);
fbAutoSineMotion(
    fPosition := fbEncoderScaling.fNormalizedPosition,
    bStartPosOK := bStartPosOK,
    bAutoEnable := bAutoEnable,
    fSineReferenceSignal := _w1); // FB_AutoSineMotion
G_Motion_Control.fWinchValveNormalizedInput_sine := fbAutoSineMotion.fWinchValveNormalizedInput;

// NETWORK 7
fbClock_dis(bEnable := bAutoEnable AND G_Engineer_HMI.bSineDisplacement); // FB_Clock
F_SineFunction_secondary(fTime := fbClock_dis.fTime, fSineSignal => _w2);
fbDisplacementControl(
    bEnable := bAutoEnable AND G_Engineer_HMI.bSineDisplacement,
    fDisplacementNormalizedInput := _w2,
    fYokeNormalizedFeedback := G_Sensors.fYokeNormalizedFeedback); // FB_DisplacementControl
G_Motion_Control.fDisplacementControlSignal_sine := fbDisplacementControl.fNormalizedOutput;

// NETWORK 8
fbJoystick(
    bEnable := bManualEnable,
    fNormalizedInput := G_Sensors.fJoystickNormalizedY,
    stParam := G_Parameters.stParam); // FB_Joystick
fWinchVelRefManual := fbJoystick.fOuput;

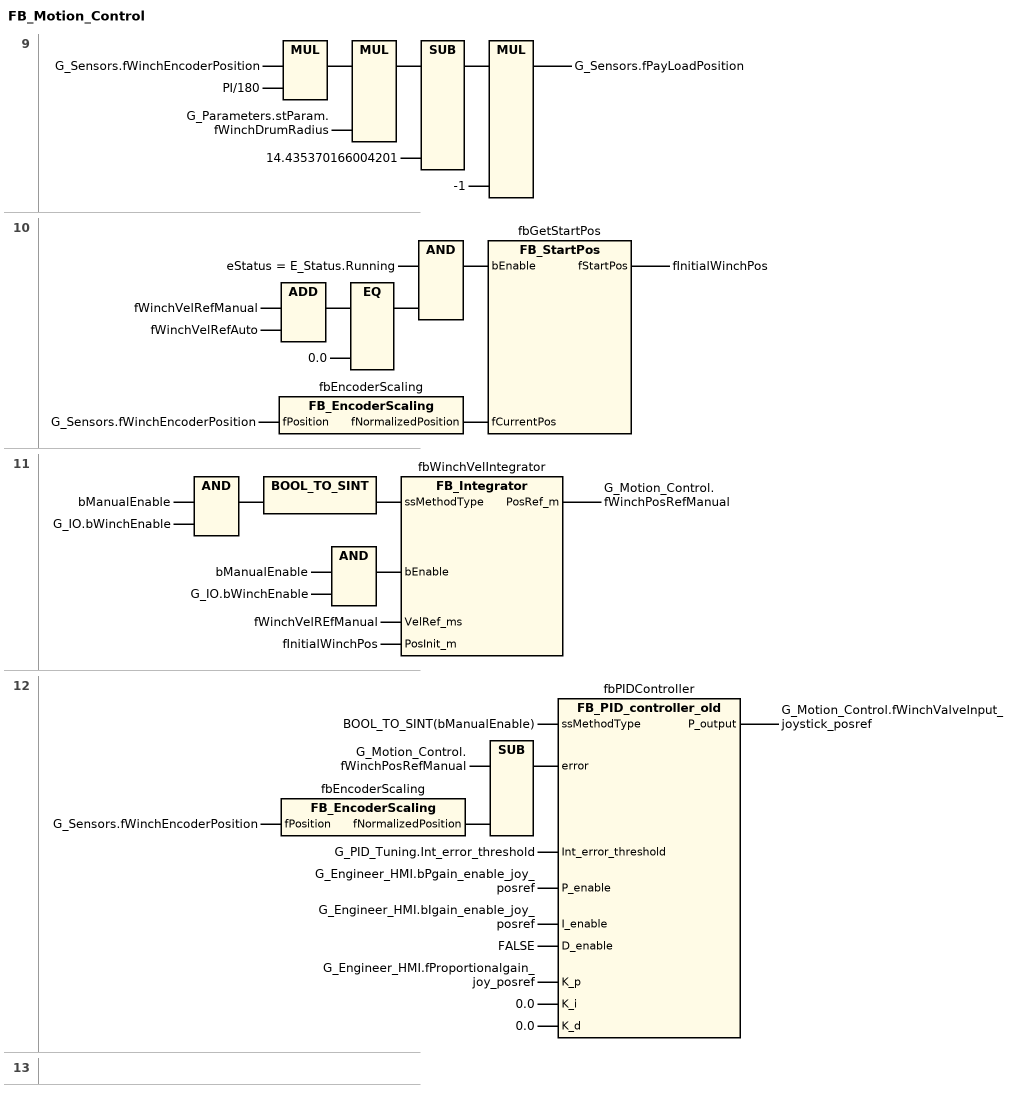
// NETWORK 9
G_Sensors.fPayLoadPosition := ((G_Sensors.fWinchEncoderPosition * (PI/180)) * G_Parameters.stParam.fWinchDrumRadius - 14.435370166004201) * -1;

// NETWORK 10
fbEncoderScaling(fPosition := G_Sensors.fWinchEncoderPosition); // FB_EncoderScaling
fbGetStartPos(bEnable := (eStatus = E_Status.Running) AND fWinchVelRefManual + fWinchVelRefAuto = 0.0, fCurrentPos := fbEncoderScaling.fNormalizedPosition); // FB_StartPos
fInitialWinchPos := fbGetStartPos.fStartPos;

// NETWORK 11
fbWinchVelIntegrator(
    ssMethodType := BOOL_TO_SINT(bManualEnable AND G_IO.bWinchEnable),
    bEnable := bManualEnable AND G_IO.bWinchEnable,
    VelRef_ms := fWinchVelREfManual,
    PosInit_m := fInitialWinchPos); // FB_Integrator
G_Motion_Control.fWinchPosRefManual := fbWinchVelIntegrator.PosRef_m;

// NETWORK 12
fbEncoderScaling(fPosition := G_Sensors.fWinchEncoderPosition); // FB_EncoderScaling
fbPIDController(
    ssMethodType := BOOL_TO_SINT(bManualEnable),
    error := G_Motion_Control.fWinchPosRefManual - fbEncoderScaling.fNormalizedPosition,
    Int_error_threshold := G_PID_Tuning.Int_error_threshold,
    P_enable := G_Engineer_HMI.bPgain_enable_joy_posref,
    I_enable := G_Engineer_HMI.bIgain_enable_joy_posref,
    D_enable := FALSE,
    K_p := G_Engineer_HMI.fProportionalgain_joy_posref,
    K_i := 0.0,
    K_d := 0.0); // FB_PID_controller_old
G_Motion_Control.fWinchValveInput_joystick_posref := fbPIDController.P_output;

// NETWORK 13

END_FUNCTION_BLOCK

// ---- Function Blocks/Currently not in use/FB_SecondaryControlStartPos.TcPOU
FUNCTION_BLOCK FB_SecondaryControlStartPos
VAR_INPUT
	bEnable 						: BOOL; 
	fPosition						: LREAL;
	fStartPosition					: LREAL;
	
	eStatus 						: BOOL; //E_Status;
END_VAR
VAR_OUTPUT
	bStartPosOK						: BOOL;
	fDisplacementControlSignal		: LREAL;
	bOpenBreak						: BOOL;
END_VAR
VAR PERSISTENT
	fProportionalGain 				: LREAL;
	fIntegralGain					: LREAL;
	fDerivateGain					: LREAL;
END_VAR
VAR
	fbPID_controller				: FB_PID_controller_old;
	fPosition_error					: LREAL;
	fProportinalGain_output			: LREAL;
	fIntegralGain_output			: LREAL;
	fDerivateGain_output			: LREAL;
    bEnableValveOutputDisp			: BOOL;	
END_VAR

IF eStatus AND G_Engineer_HMI.bSecondaryStartPosEnable THEN
	bOpenBreak	:= TRUE;
ELSE
	bOpenBreak := FALSE;
END_IF

IF bEnable THEN 
	
fPosition_error := fStartPosition - fPosition;

G_Motion_Control.fPosition_error_StartDisplacement := fPosition_error; 

